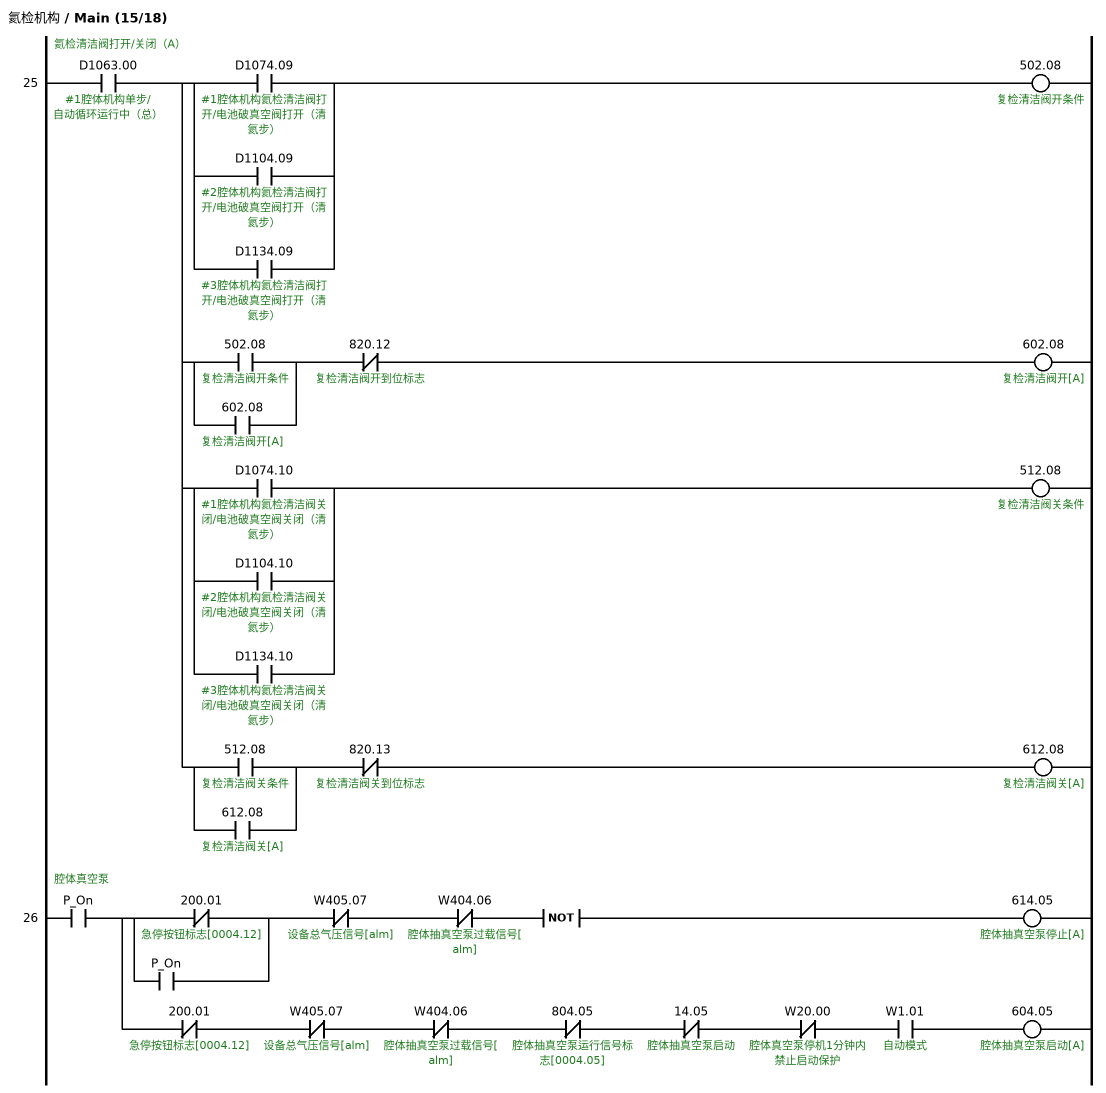
; [picture p144: 氦检机构 / Main, rungs 25-26]
; rung 25: 氦检清洁阀打开/关闭（A）
LD D1063.00  ; #1腔体机构单步/自动循环运行中（总）
OUT TR0
LD D1074.09  ; #1腔体机构氦检清洁阀打开/电池破真空阀打开（清氦步）
OR D1104.09  ; #2腔体机构氦检清洁阀打开/电池破真空阀打开（清氦步）
OR D1134.09  ; #3腔体机构氦检清洁阀打开/电池破真空阀打开（清氦步）
ANDLD
OUT 502.08  ; 复检清洁阀开条件
LD TR0
LD 502.08  ; 复检清洁阀开条件
OR 602.08  ; 复检清洁阀开[A]
ANDLD
ANDNOT 820.12  ; 复检清洁阀开到位标志
OUT 602.08  ; 复检清洁阀开[A]
LD TR0
LD D1074.10  ; #1腔体机构氦检清洁阀关闭/电池破真空阀关闭（清氦步）
OR D1104.10  ; #2腔体机构氦检清洁阀关闭/电池破真空阀关闭（清氦步）
OR D1134.10  ; #3腔体机构氦检清洁阀关闭/电池破真空阀关闭（清氦步）
ANDLD
OUT 512.08  ; 复检清洁阀关条件
LD TR0
LD 512.08  ; 复检清洁阀关条件
OR 612.08  ; 复检清洁阀关[A]
ANDLD
ANDNOT 820.13  ; 复检清洁阀关到位标志
OUT 612.08  ; 复检清洁阀关[A]
; rung 26: 腔体真空泵
LD P_On
OUT TR0
LDNOT 200.01  ; 急停按钮标志[0004.12]
OR P_On
ANDLD
ANDNOT W405.07  ; 设备总气压信号[alm]
ANDNOT W404.06  ; 腔体抽真空泵过载信号[alm]
NOT(520)
OUT 614.05  ; 腔体抽真空泵停止[A]
LD TR0
ANDNOT 200.01  ; 急停按钮标志[0004.12]
ANDNOT W405.07  ; 设备总气压信号[alm]
ANDNOT W404.06  ; 腔体抽真空泵过载信号[alm]
ANDNOT 804.05  ; 腔体抽真空泵运行信号标志[0004.05]
ANDNOT 14.05  ; 腔体抽真空泵启动
ANDNOT W20.00  ; 腔体真空泵停机1分钟内禁止启动保护
AND W1.01  ; 自动模式
OUT 604.05  ; 腔体抽真空泵启动[A]

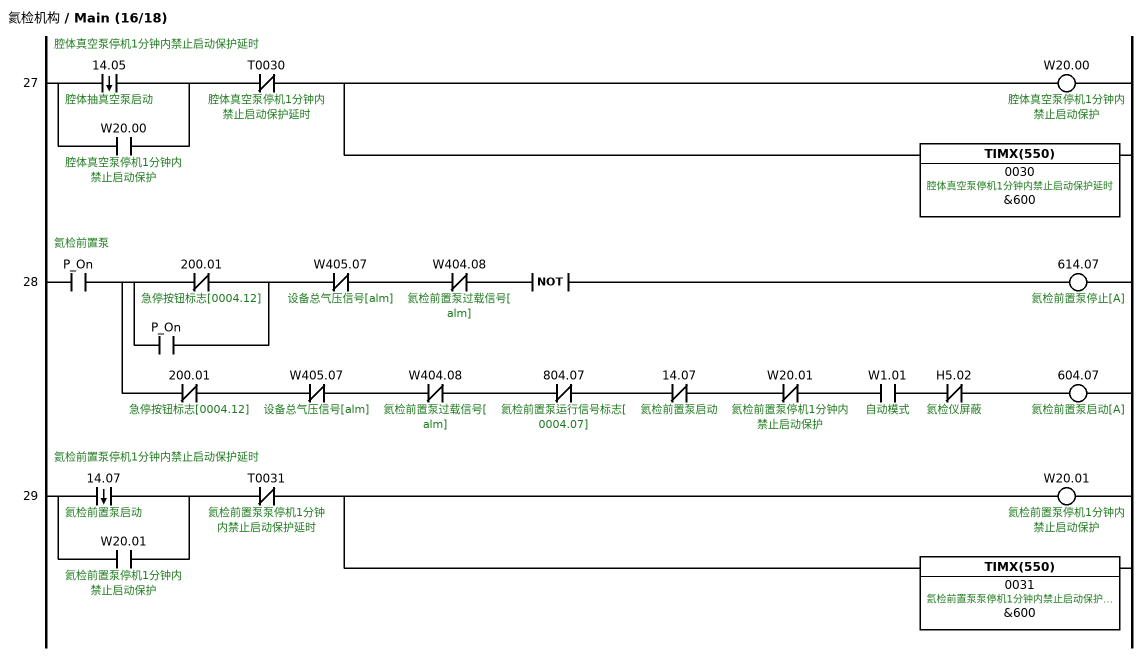
; rung 27: 腔体真空泵停机1分钟内禁止启动保护延时
%LD 14.05  ; 腔体抽真空泵启动
OR W20.00  ; 腔体真空泵停机1分钟内禁止启动保护
ANDNOT T0030  ; 腔体真空泵停机1分钟内禁止启动保护延时
OUT W20.00  ; 腔体真空泵停机1分钟内禁止启动保护
TIMX(550) 0030 &600  ; 腔体真空泵停机1分钟内禁止启动保护延时
; rung 28: 氦检前置泵
LD P_On
OUT TR0
LDNOT 200.01  ; 急停按钮标志[0004.12]
OR P_On
ANDLD
ANDNOT W405.07  ; 设备总气压信号[alm]
ANDNOT W404.08  ; 氦检前置泵过载信号[alm]
NOT(520)
OUT 614.07  ; 氦检前置泵停止[A]
LD TR0
ANDNOT 200.01  ; 急停按钮标志[0004.12]
ANDNOT W405.07  ; 设备总气压信号[alm]
ANDNOT W404.08  ; 氦检前置泵过载信号[alm]
ANDNOT 804.07  ; 氦检前置泵运行信号标志[0004.07]
ANDNOT 14.07  ; 氦检前置泵启动
ANDNOT W20.01  ; 氦检前置泵停机1分钟内禁止启动保护
AND W1.01  ; 自动模式
ANDNOT H5.02  ; 氦检仪屏蔽
OUT 604.07  ; 氦检前置泵启动[A]
; rung 29: 氦检前置泵停机1分钟内禁止启动保护延时
%LD 14.07  ; 氦检前置泵启动
OR W20.01  ; 氦检前置泵停机1分钟内禁止启动保护
ANDNOT T0031  ; 氦检前置泵泵停机1分钟内禁止启动保护延时
OUT W20.01  ; 氦检前置泵停机1分钟内禁止启动保护
TIMX(550) 0031 &600  ; 氦检前置泵泵停机1分钟内禁止启动保护延时

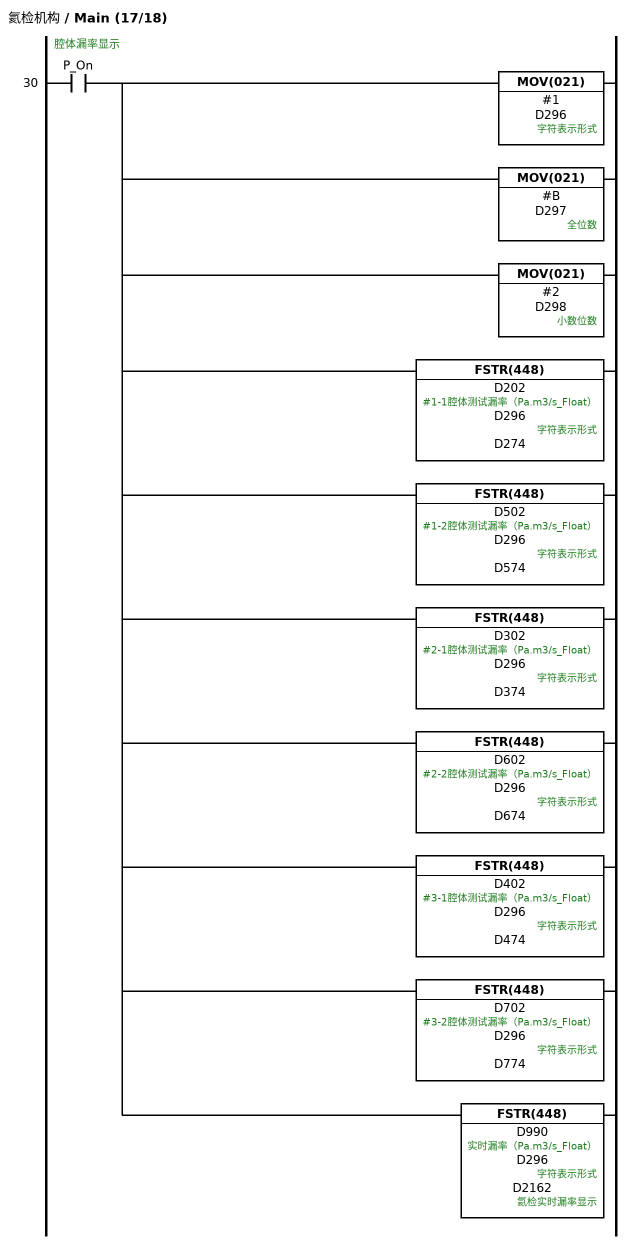
; rung 30: 腔体漏率显示
LD P_On
MOV(021) #1 D296  ; 字符表示形式
MOV(021) #B D297  ; 全位数
MOV(021) #2 D298  ; 小数位数
FSTR(448) D202 D296 D274  ; #1-1腔体测试漏率（Pa.m3/s_Float）, 字符表示形式
FSTR(448) D502 D296 D574  ; #1-2腔体测试漏率（Pa.m3/s_Float）, 字符表示形式
FSTR(448) D302 D296 D374  ; #2-1腔体测试漏率（Pa.m3/s_Float）, 字符表示形式
FSTR(448) D602 D296 D674  ; #2-2腔体测试漏率（Pa.m3/s_Float）, 字符表示形式
FSTR(448) D402 D296 D474  ; #3-1腔体测试漏率（Pa.m3/s_Float）, 字符表示形式
FSTR(448) D702 D296 D774  ; #3-2腔体测试漏率（Pa.m3/s_Float）, 字符表示形式
FSTR(448) D990 D296 D2162  ; 实时漏率（Pa.m3/s_Float）, 字符表示形式, 氦检实时漏率显示

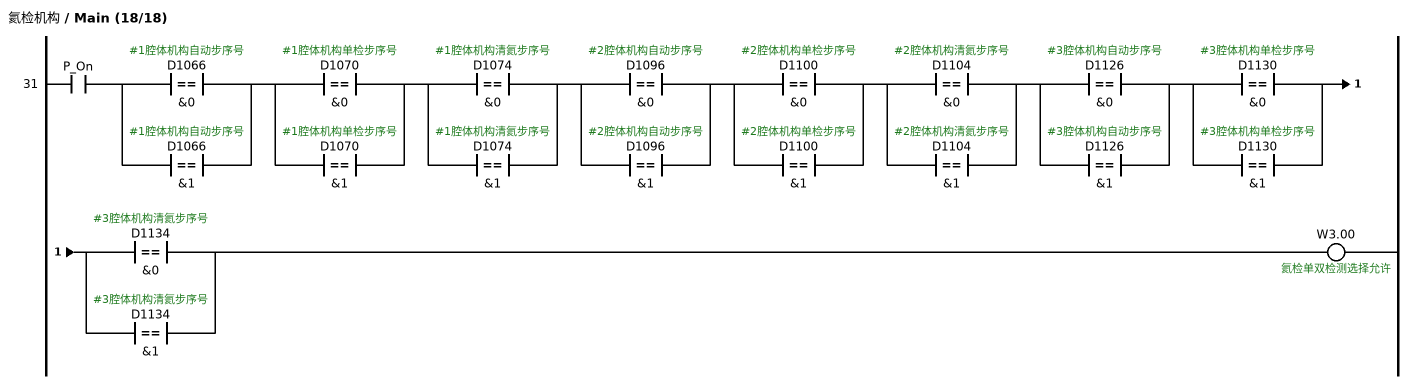
; rung 31
LD P_On
LD=L(301) D1066 &0  ; #1腔体机构自动步序号
OR=L(301) D1066 &1  ; #1腔体机构自动步序号
ANDLD
LD=L(301) D1070 &0  ; #1腔体机构单检步序号
OR=L(301) D1070 &1  ; #1腔体机构单检步序号
ANDLD
LD=L(301) D1074 &0  ; #1腔体机构清氦步序号
OR=L(301) D1074 &1  ; #1腔体机构清氦步序号
ANDLD
LD=L(301) D1096 &0  ; #2腔体机构自动步序号
OR=L(301) D1096 &1  ; #2腔体机构自动步序号
ANDLD
LD=L(301) D1100 &0  ; #2腔体机构单检步序号
OR=L(301) D1100 &1  ; #2腔体机构单检步序号
ANDLD
LD=L(301) D1104 &0  ; #2腔体机构清氦步序号
OR=L(301) D1104 &1  ; #2腔体机构清氦步序号
ANDLD
LD=L(301) D1126 &0  ; #3腔体机构自动步序号
OR=L(301) D1126 &1  ; #3腔体机构自动步序号
ANDLD
LD=L(301) D1130 &0  ; #3腔体机构单检步序号
OR=L(301) D1130 &1  ; #3腔体机构单检步序号
ANDLD
LD=L(301) D1134 &0  ; #3腔体机构清氦步序号
OR=L(301) D1134 &1  ; #3腔体机构清氦步序号
ANDLD
OUT W3.00  ; 氦检单双检测选择允许

### Section 氦检腔1手动

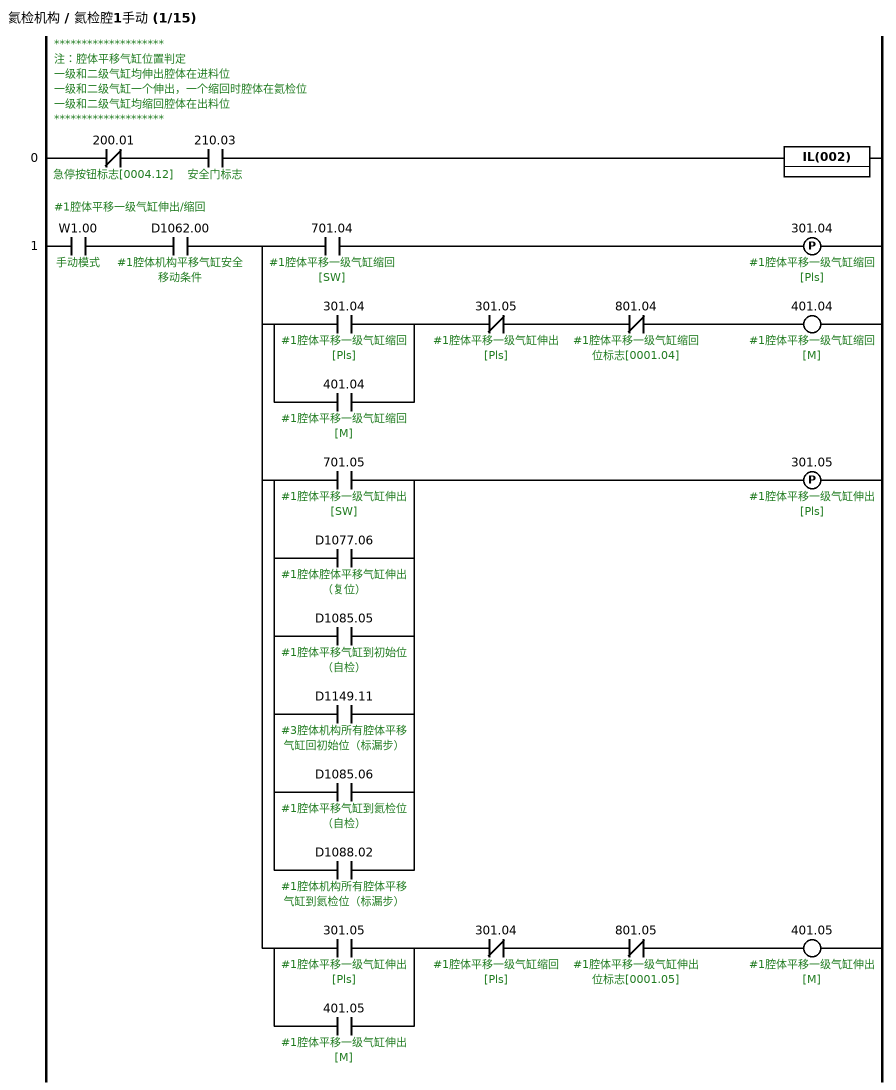
; rung 0: ******************** / 注：腔体平移气缸位置判定 / 一级和二级气缸均伸出腔体在进料位 / 一级和二级气缸一个伸出，一个缩回时腔体在氦检位 / 一级和二级气缸均缩回腔体在出料位 / ********************
LDNOT 200.01  ; 急停按钮标志[0004.12]
AND 210.03  ; 安全门标志
IL(002)
; rung 1: #1腔体平移一级气缸伸出/缩回
LD W1.00  ; 手动模式
AND D1062.00  ; #1腔体机构平移气缸安全移动条件
OUT TR0
AND 701.04  ; #1腔体平移一级气缸缩回[SW]
DIFU(013) 301.04  ; #1腔体平移一级气缸缩回[Pls]
LD TR0
LD 301.04  ; #1腔体平移一级气缸缩回[Pls]
OR 401.04  ; #1腔体平移一级气缸缩回[M]
ANDLD
ANDNOT 301.05  ; #1腔体平移一级气缸伸出[Pls]
ANDNOT 801.04  ; #1腔体平移一级气缸缩回位标志[0001.04]
OUT 401.04  ; #1腔体平移一级气缸缩回[M]
LD TR0
LD 701.05  ; #1腔体平移一级气缸伸出[SW]
OR D1077.06  ; #1腔体腔体平移气缸伸出（复位）
OR D1085.05  ; #1腔体平移气缸到初始位（自检）
OR D1149.11  ; #3腔体机构所有腔体平移气缸回初始位（标漏步）
OR D1085.06  ; #1腔体平移气缸到氦检位（自检）
OR D1088.02  ; #1腔体机构所有腔体平移气缸到氦检位（标漏步）
ANDLD
DIFU(013) 301.05  ; #1腔体平移一级气缸伸出[Pls]
LD TR0
LD 301.05  ; #1腔体平移一级气缸伸出[Pls]
OR 401.05  ; #1腔体平移一级气缸伸出[M]
ANDLD
ANDNOT 301.04  ; #1腔体平移一级气缸缩回[Pls]
ANDNOT 801.05  ; #1腔体平移一级气缸伸出位标志[0001.05]
OUT 401.05  ; #1腔体平移一级气缸伸出[M]

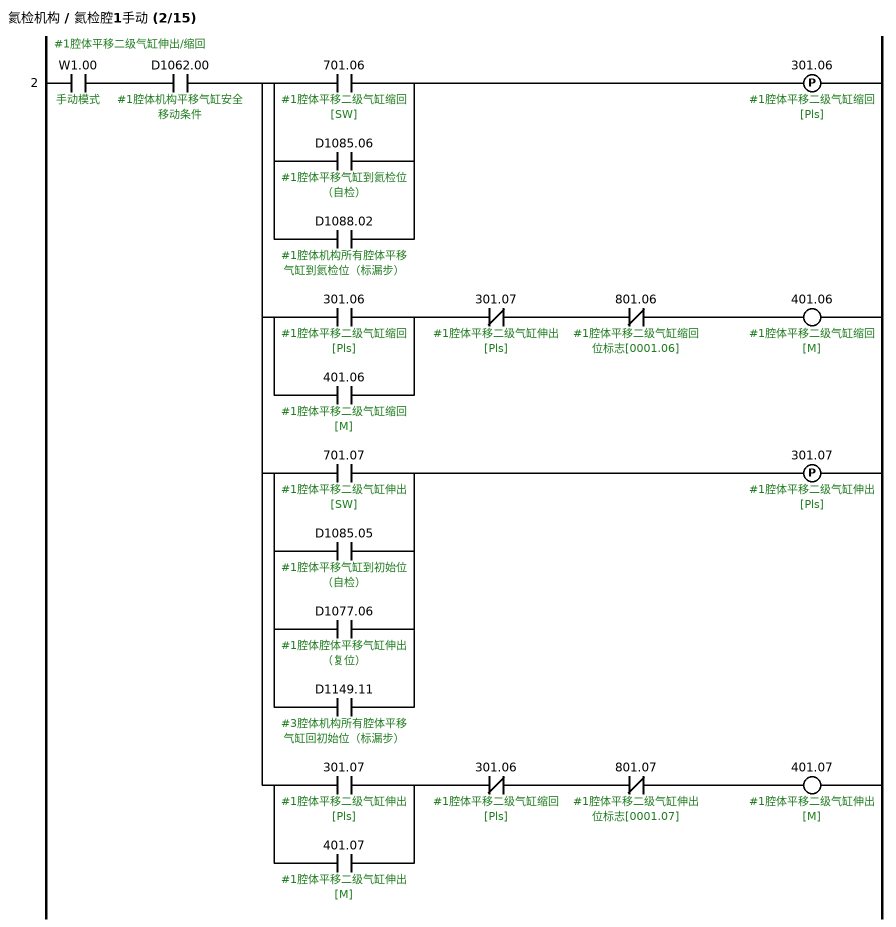
; rung 2: #1腔体平移二级气缸伸出/缩回
LD W1.00  ; 手动模式
AND D1062.00  ; #1腔体机构平移气缸安全移动条件
OUT TR0
LD 701.06  ; #1腔体平移二级气缸缩回[SW]
OR D1085.06  ; #1腔体平移气缸到氦检位（自检）
OR D1088.02  ; #1腔体机构所有腔体平移气缸到氦检位（标漏步）
ANDLD
DIFU(013) 301.06  ; #1腔体平移二级气缸缩回[Pls]
LD TR0
LD 301.06  ; #1腔体平移二级气缸缩回[Pls]
OR 401.06  ; #1腔体平移二级气缸缩回[M]
ANDLD
ANDNOT 301.07  ; #1腔体平移二级气缸伸出[Pls]
ANDNOT 801.06  ; #1腔体平移二级气缸缩回位标志[0001.06]
OUT 401.06  ; #1腔体平移二级气缸缩回[M]
LD TR0
LD 701.07  ; #1腔体平移二级气缸伸出[SW]
OR D1085.05  ; #1腔体平移气缸到初始位（自检）
OR D1077.06  ; #1腔体腔体平移气缸伸出（复位）
OR D1149.11  ; #3腔体机构所有腔体平移气缸回初始位（标漏步）
ANDLD
DIFU(013) 301.07  ; #1腔体平移二级气缸伸出[Pls]
LD TR0
LD 301.07  ; #1腔体平移二级气缸伸出[Pls]
OR 401.07  ; #1腔体平移二级气缸伸出[M]
ANDLD
ANDNOT 301.06  ; #1腔体平移二级气缸缩回[Pls]
ANDNOT 801.07  ; #1腔体平移二级气缸伸出位标志[0001.07]
OUT 401.07  ; #1腔体平移二级气缸伸出[M]

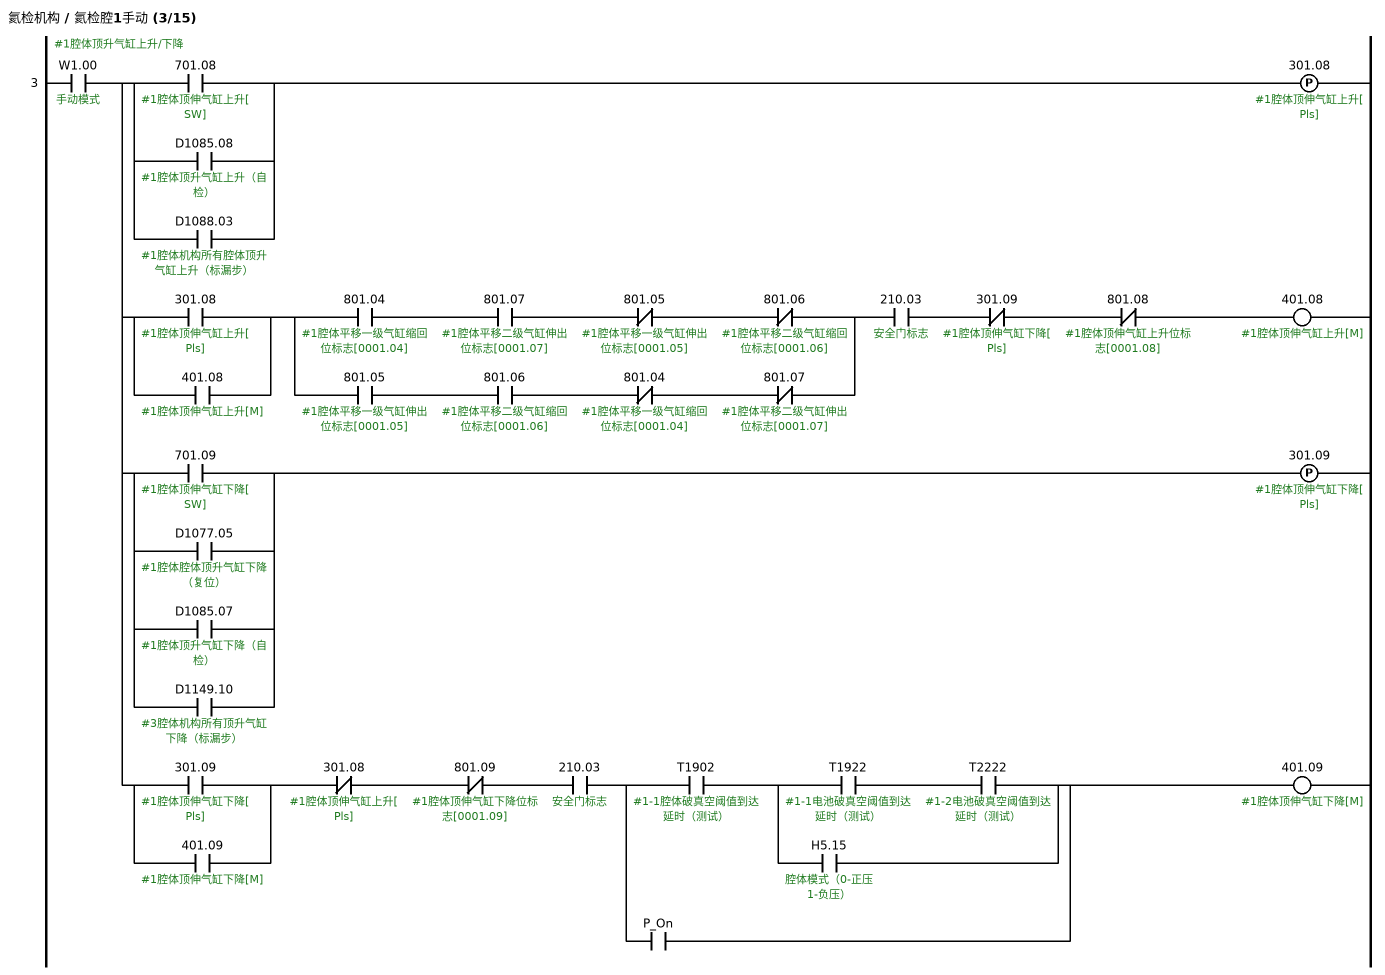
; rung 3: #1腔体顶升气缸上升/下降
LD W1.00  ; 手动模式
OUT TR0
LD 701.08  ; #1腔体顶伸气缸上升[SW]
OR D1085.08  ; #1腔体顶升气缸上升（自检）
OR D1088.03  ; #1腔体机构所有腔体顶升气缸上升（标漏步）
ANDLD
DIFU(013) 301.08  ; #1腔体顶伸气缸上升[Pls]
LD TR0
LD 301.08  ; #1腔体顶伸气缸上升[Pls]
OR 401.08  ; #1腔体顶伸气缸上升[M]
ANDLD
LD 801.04  ; #1腔体平移一级气缸缩回位标志[0001.04]
AND 801.07  ; #1腔体平移二级气缸伸出位标志[0001.07]
ANDNOT 801.05  ; #1腔体平移一级气缸伸出位标志[0001.05]
ANDNOT 801.06  ; #1腔体平移二级气缸缩回位标志[0001.06]
LD 801.05  ; #1腔体平移一级气缸伸出位标志[0001.05]
AND 801.06  ; #1腔体平移二级气缸缩回位标志[0001.06]
ANDNOT 801.04  ; #1腔体平移一级气缸缩回位标志[0001.04]
ANDNOT 801.07  ; #1腔体平移二级气缸伸出位标志[0001.07]
ORLD
ANDLD
AND 210.03  ; 安全门标志
ANDNOT 301.09  ; #1腔体顶伸气缸下降[Pls]
ANDNOT 801.08  ; #1腔体顶伸气缸上升位标志[0001.08]
OUT 401.08  ; #1腔体顶伸气缸上升[M]
LD TR0
LD 701.09  ; #1腔体顶伸气缸下降[SW]
OR D1077.05  ; #1腔体腔体顶升气缸下降（复位）
OR D1085.07  ; #1腔体顶升气缸下降（自检）
OR D1149.10  ; #3腔体机构所有顶升气缸下降（标漏步）
ANDLD
DIFU(013) 301.09  ; #1腔体顶伸气缸下降[Pls]
LD TR0
LD 301.09  ; #1腔体顶伸气缸下降[Pls]
OR 401.09  ; #1腔体顶伸气缸下降[M]
ANDLD
ANDNOT 301.08  ; #1腔体顶伸气缸上升[Pls]
ANDNOT 801.09  ; #1腔体顶伸气缸下降位标志[0001.09]
AND 210.03  ; 安全门标志
LD T1902  ; #1-1腔体破真空阈值到达延时（测试）
LD T1922  ; #1-1电池破真空阈值到达延时（测试）
AND T2222  ; #1-2电池破真空阈值到达延时（测试）
OR H5.15  ; 腔体模式（0-正压 1-负压）
ANDLD
OR P_On
ANDLD
OUT 401.09  ; #1腔体顶伸气缸下降[M]

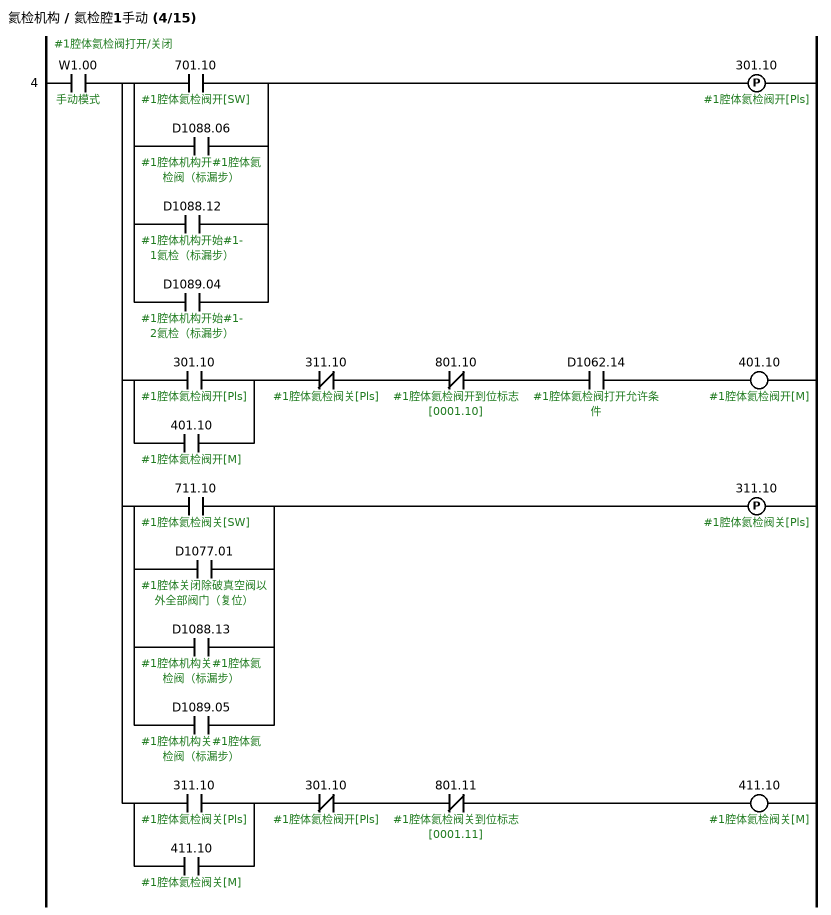
; rung 4: #1腔体氦检阀打开/关闭
LD W1.00  ; 手动模式
OUT TR0
LD 701.10  ; #1腔体氦检阀开[SW]
OR D1088.06  ; #1腔体机构开#1腔体氦检阀（标漏步）
OR D1088.12  ; #1腔体机构开始#1-1氦检（标漏步）
OR D1089.04  ; #1腔体机构开始#1-2氦检（标漏步）
ANDLD
DIFU(013) 301.10  ; #1腔体氦检阀开[Pls]
LD TR0
LD 301.10  ; #1腔体氦检阀开[Pls]
OR 401.10  ; #1腔体氦检阀开[M]
ANDLD
ANDNOT 311.10  ; #1腔体氦检阀关[Pls]
ANDNOT 801.10  ; #1腔体氦检阀开到位标志[0001.10]
AND D1062.14  ; #1腔体氦检阀打开允许条件
OUT 401.10  ; #1腔体氦检阀开[M]
LD TR0
LD 711.10  ; #1腔体氦检阀关[SW]
OR D1077.01  ; #1腔体关闭除破真空阀以外全部阀门（复位）
OR D1088.13  ; #1腔体机构关#1腔体氦检阀（标漏步）
OR D1089.05  ; #1腔体机构关#1腔体氦检阀（标漏步）
ANDLD
DIFU(013) 311.10  ; #1腔体氦检阀关[Pls]
LD TR0
LD 311.10  ; #1腔体氦检阀关[Pls]
OR 411.10  ; #1腔体氦检阀关[M]
ANDLD
ANDNOT 301.10  ; #1腔体氦检阀开[Pls]
ANDNOT 801.11  ; #1腔体氦检阀关到位标志[0001.11]
OUT 411.10  ; #1腔体氦检阀关[M]

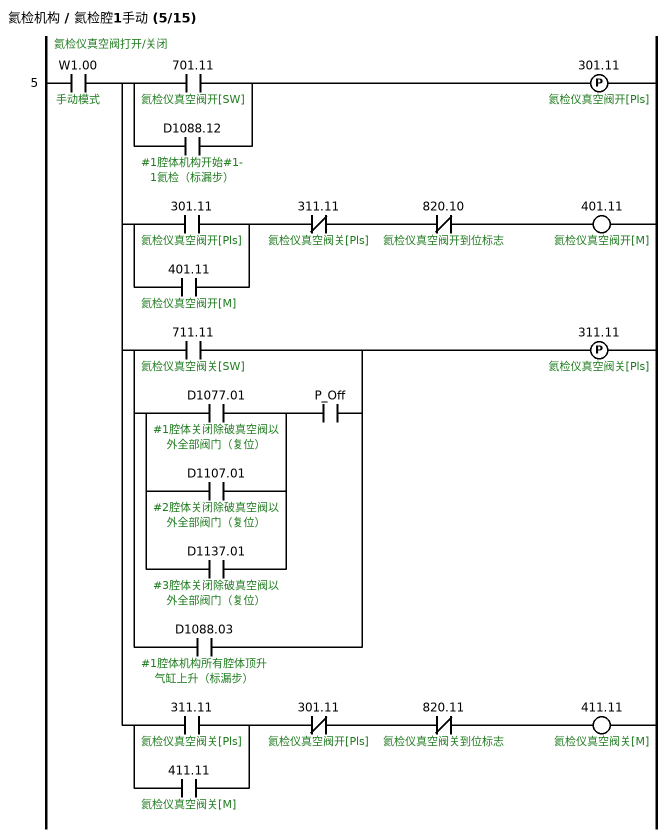
; rung 5: 氦检仪真空阀打开/关闭
LD W1.00  ; 手动模式
OUT TR0
LD 701.11  ; 氦检仪真空阀开[SW]
OR D1088.12  ; #1腔体机构开始#1-1氦检（标漏步）
ANDLD
DIFU(013) 301.11  ; 氦检仪真空阀开[Pls]
LD TR0
LD 301.11  ; 氦检仪真空阀开[Pls]
OR 401.11  ; 氦检仪真空阀开[M]
ANDLD
ANDNOT 311.11  ; 氦检仪真空阀关[Pls]
ANDNOT 820.10  ; 氦检仪真空阀开到位标志
OUT 401.11  ; 氦检仪真空阀开[M]
LD TR0
LD 711.11  ; 氦检仪真空阀关[SW]
LD D1077.01  ; #1腔体关闭除破真空阀以外全部阀门（复位）
OR D1107.01  ; #2腔体关闭除破真空阀以外全部阀门（复位）
OR D1137.01  ; #3腔体关闭除破真空阀以外全部阀门（复位）
AND P_Off
ORLD
OR D1088.03  ; #1腔体机构所有腔体顶升气缸上升（标漏步）
ANDLD
DIFU(013) 311.11  ; 氦检仪真空阀关[Pls]
LD TR0
LD 311.11  ; 氦检仪真空阀关[Pls]
OR 411.11  ; 氦检仪真空阀关[M]
ANDLD
ANDNOT 301.11  ; 氦检仪真空阀开[Pls]
ANDNOT 820.11  ; 氦检仪真空阀关到位标志
OUT 411.11  ; 氦检仪真空阀关[M]

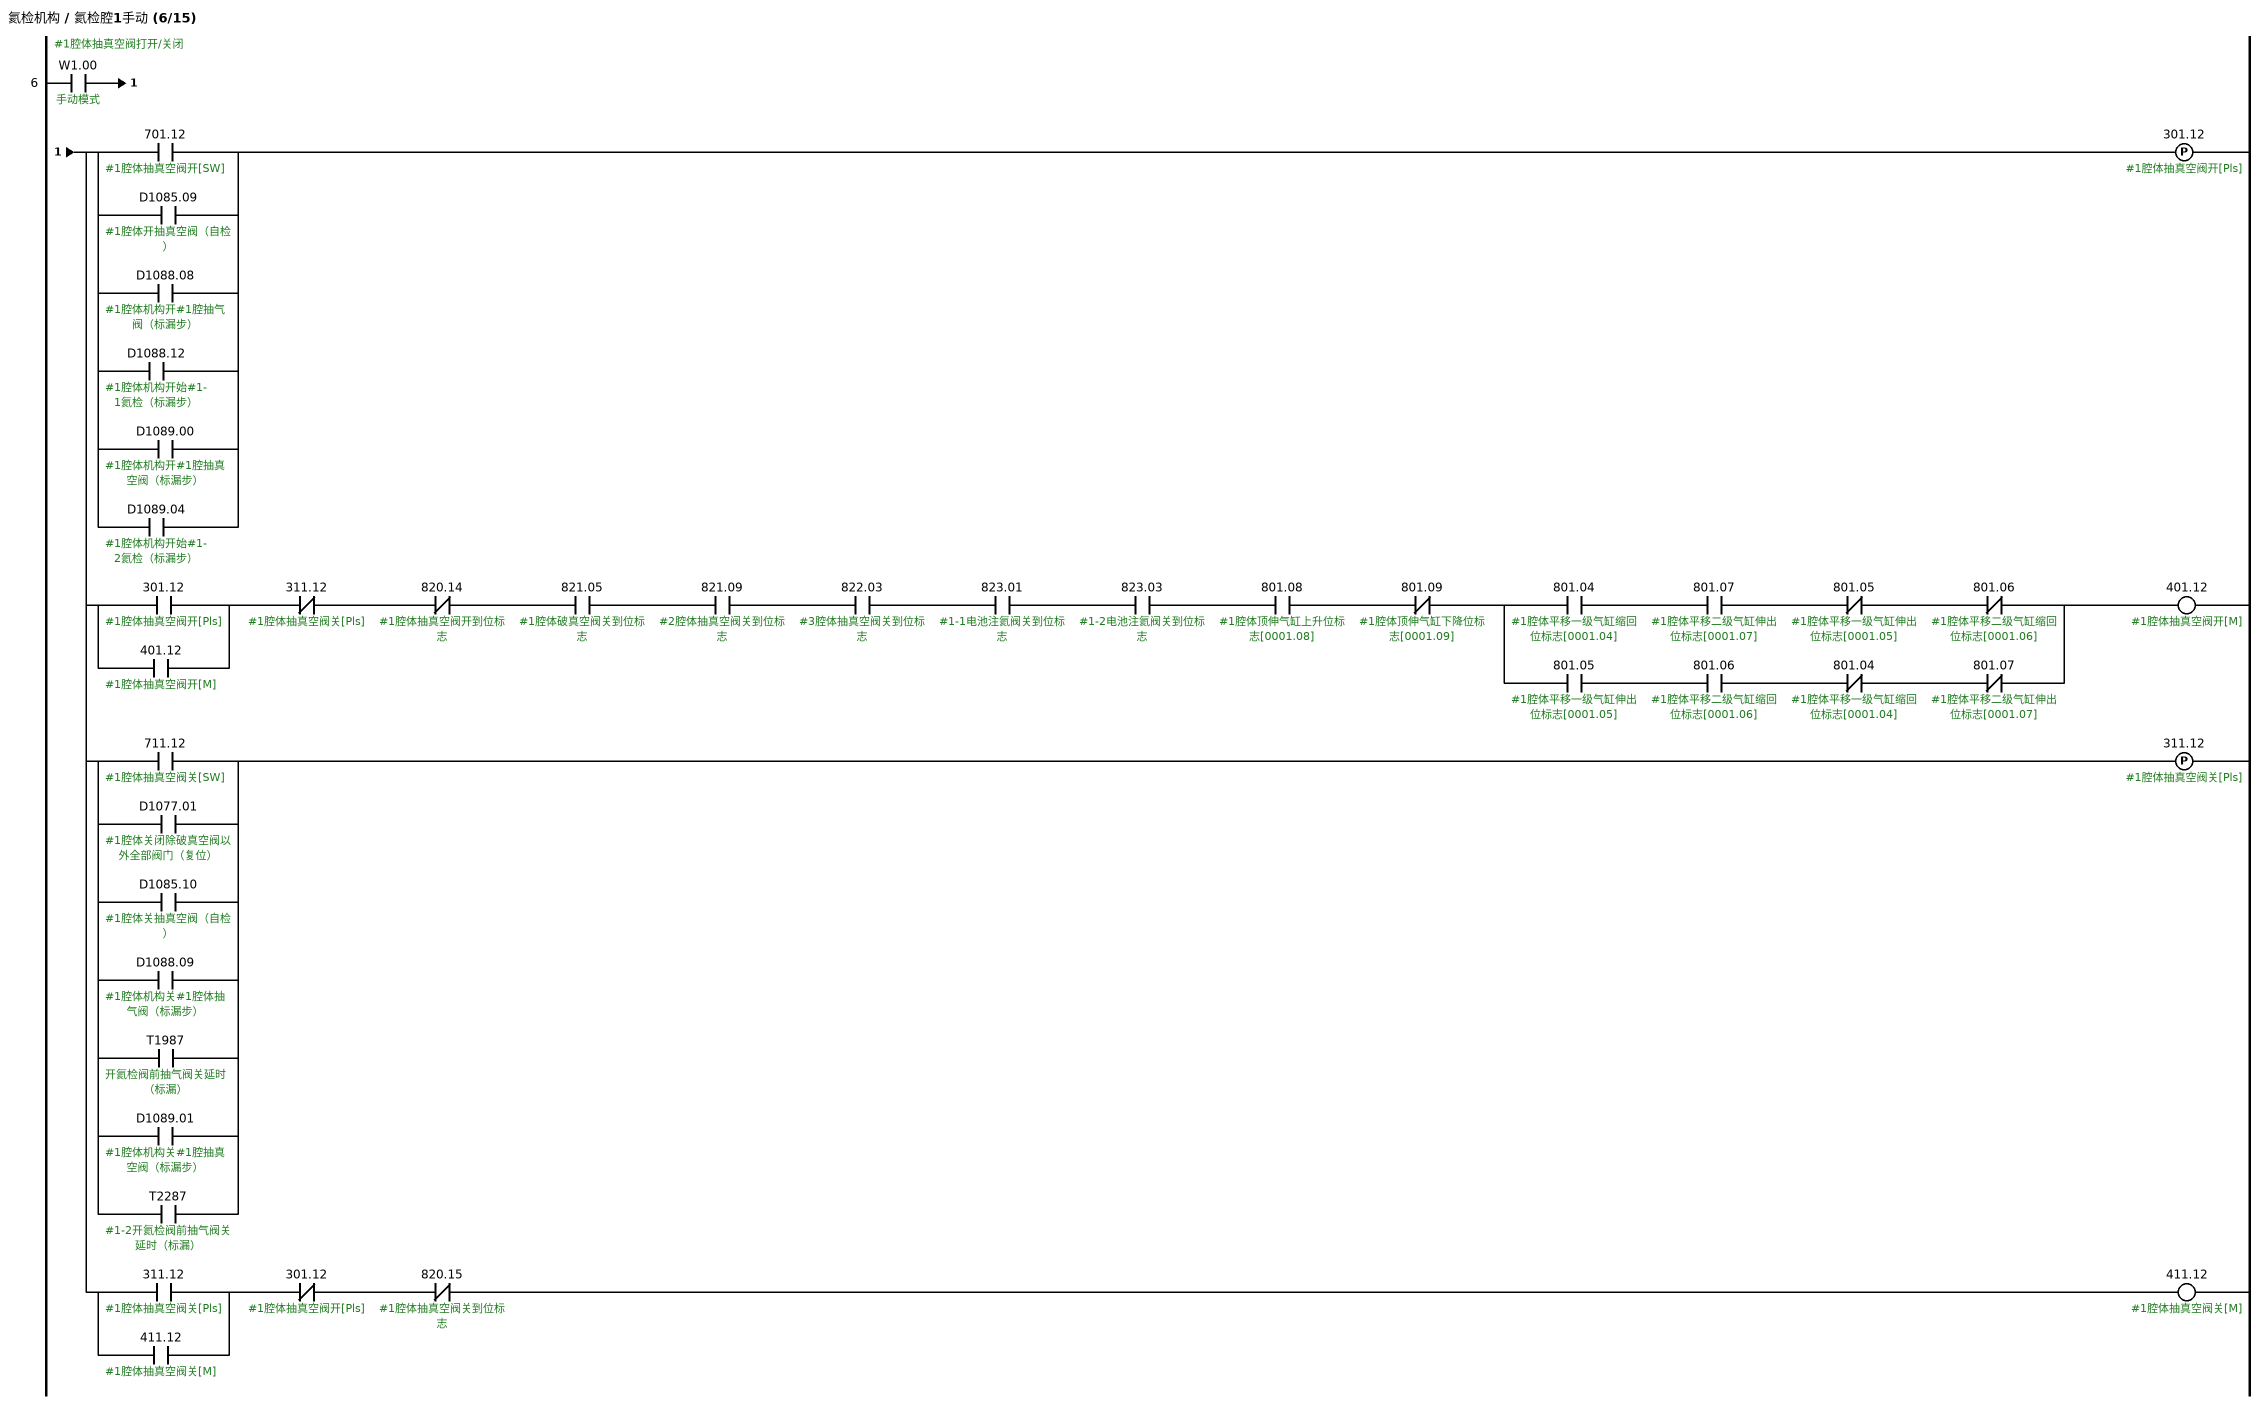
; rung 6: #1腔体抽真空阀打开/关闭
LD W1.00  ; 手动模式
OUT TR0
LD 701.12  ; #1腔体抽真空阀开[SW]
OR D1085.09  ; #1腔体开抽真空阀（自检）
OR D1088.08  ; #1腔体机构开#1腔抽气阀（标漏步）
OR D1088.12  ; #1腔体机构开始#1-1氦检（标漏步）
OR D1089.00  ; #1腔体机构开#1腔抽真空阀（标漏步）
OR D1089.04  ; #1腔体机构开始#1-2氦检（标漏步）
ANDLD
DIFU(013) 301.12  ; #1腔体抽真空阀开[Pls]
LD TR0
LD 301.12  ; #1腔体抽真空阀开[Pls]
OR 401.12  ; #1腔体抽真空阀开[M]
ANDLD
ANDNOT 311.12  ; #1腔体抽真空阀关[Pls]
ANDNOT 820.14  ; #1腔体抽真空阀开到位标志
AND 821.05  ; #1腔体破真空阀关到位标志
AND 821.09  ; #2腔体抽真空阀关到位标志
AND 822.03  ; #3腔体抽真空阀关到位标志
AND 823.01  ; #1-1电池注氦阀关到位标志
AND 823.03  ; #1-2电池注氦阀关到位标志
AND 801.08  ; #1腔体顶伸气缸上升位标志[0001.08]
ANDNOT 801.09  ; #1腔体顶伸气缸下降位标志[0001.09]
LD 801.04  ; #1腔体平移一级气缸缩回位标志[0001.04]
AND 801.07  ; #1腔体平移二级气缸伸出位标志[0001.07]
ANDNOT 801.05  ; #1腔体平移一级气缸伸出位标志[0001.05]
ANDNOT 801.06  ; #1腔体平移二级气缸缩回位标志[0001.06]
LD 801.05  ; #1腔体平移一级气缸伸出位标志[0001.05]
AND 801.06  ; #1腔体平移二级气缸缩回位标志[0001.06]
ANDNOT 801.04  ; #1腔体平移一级气缸缩回位标志[0001.04]
ANDNOT 801.07  ; #1腔体平移二级气缸伸出位标志[0001.07]
ORLD
ANDLD
OUT 401.12  ; #1腔体抽真空阀开[M]
LD TR0
LD 711.12  ; #1腔体抽真空阀关[SW]
OR D1077.01  ; #1腔体关闭除破真空阀以外全部阀门（复位）
OR D1085.10  ; #1腔体关抽真空阀（自检）
OR D1088.09  ; #1腔体机构关#1腔体抽气阀（标漏步）
OR T1987  ; 开氦检阀前抽气阀关延时（标漏）
OR D1089.01  ; #1腔体机构关#1腔抽真空阀（标漏步）
OR T2287  ; #1-2开氦检阀前抽气阀关延时（标漏）
ANDLD
DIFU(013) 311.12  ; #1腔体抽真空阀关[Pls]
LD TR0
LD 311.12  ; #1腔体抽真空阀关[Pls]
OR 411.12  ; #1腔体抽真空阀关[M]
ANDLD
ANDNOT 301.12  ; #1腔体抽真空阀开[Pls]
ANDNOT 820.15  ; #1腔体抽真空阀关到位标志
OUT 411.12  ; #1腔体抽真空阀关[M]

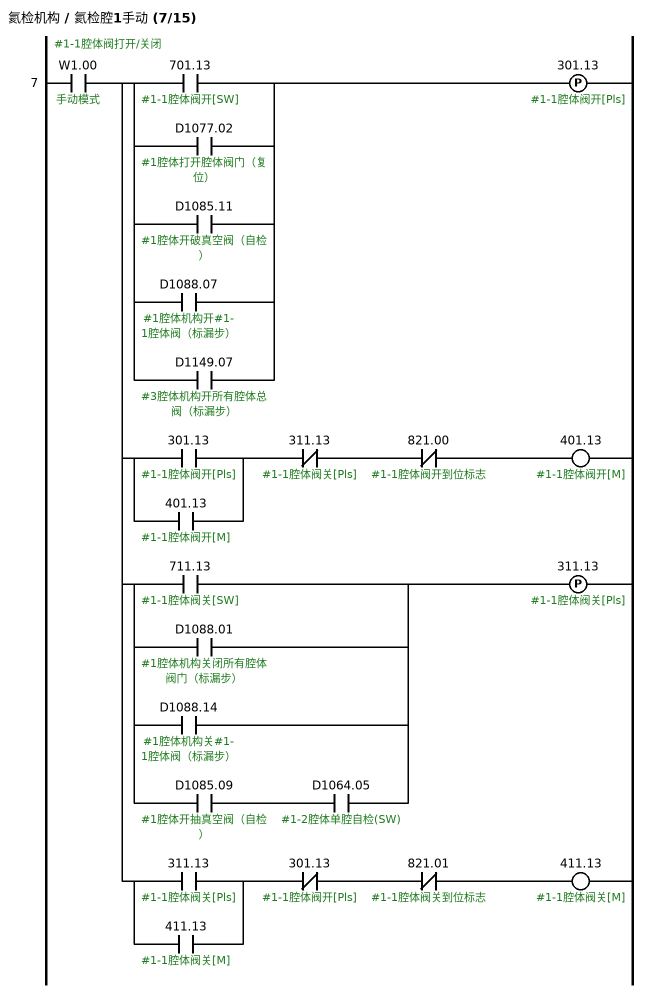
; rung 7: #1-1腔体阀打开/关闭
LD W1.00  ; 手动模式
OUT TR0
LD 701.13  ; #1-1腔体阀开[SW]
OR D1077.02  ; #1腔体打开腔体阀门（复位）
OR D1085.11  ; #1腔体开破真空阀（自检）
OR D1088.07  ; #1腔体机构开#1-1腔体阀（标漏步）
OR D1149.07  ; #3腔体机构开所有腔体总阀（标漏步）
ANDLD
DIFU(013) 301.13  ; #1-1腔体阀开[Pls]
LD TR0
LD 301.13  ; #1-1腔体阀开[Pls]
OR 401.13  ; #1-1腔体阀开[M]
ANDLD
ANDNOT 311.13  ; #1-1腔体阀关[Pls]
ANDNOT 821.00  ; #1-1腔体阀开到位标志
OUT 401.13  ; #1-1腔体阀开[M]
LD TR0
LD 711.13  ; #1-1腔体阀关[SW]
OR D1088.01  ; #1腔体机构关闭所有腔体阀门（标漏步）
OR D1088.14  ; #1腔体机构关#1-1腔体阀（标漏步）
LD D1085.09  ; #1腔体开抽真空阀（自检）
AND D1064.05  ; #1-2腔体单腔自检(SW)
ORLD
ANDLD
DIFU(013) 311.13  ; #1-1腔体阀关[Pls]
LD TR0
LD 311.13  ; #1-1腔体阀关[Pls]
OR 411.13  ; #1-1腔体阀关[M]
ANDLD
ANDNOT 301.13  ; #1-1腔体阀开[Pls]
ANDNOT 821.01  ; #1-1腔体阀关到位标志
OUT 411.13  ; #1-1腔体阀关[M]

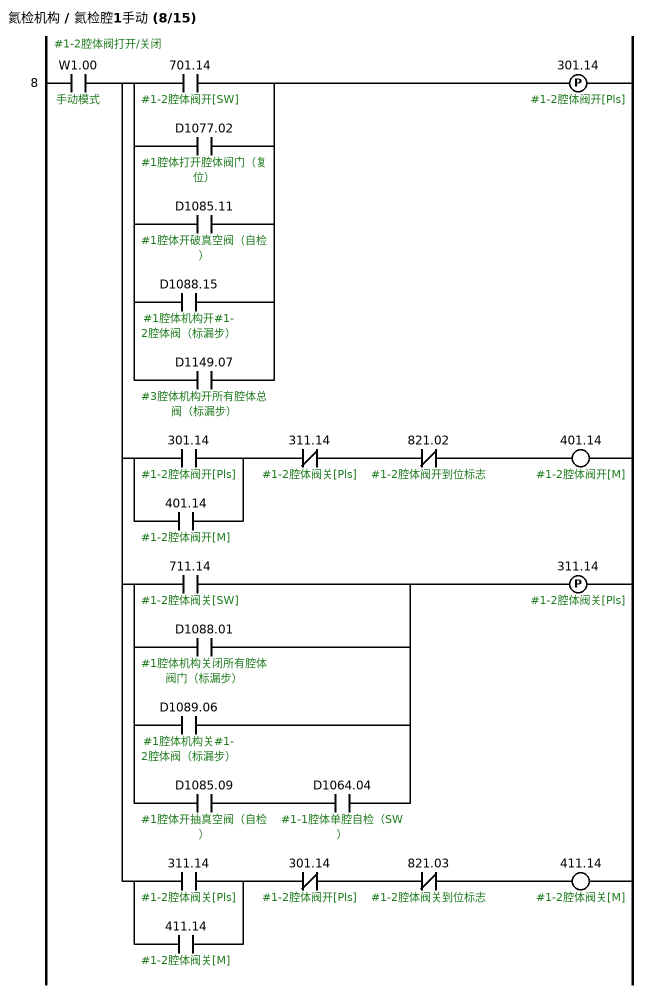
; rung 8: #1-2腔体阀打开/关闭
LD W1.00  ; 手动模式
OUT TR0
LD 701.14  ; #1-2腔体阀开[SW]
OR D1077.02  ; #1腔体打开腔体阀门（复位）
OR D1085.11  ; #1腔体开破真空阀（自检）
OR D1088.15  ; #1腔体机构开#1-2腔体阀（标漏步）
OR D1149.07  ; #3腔体机构开所有腔体总阀（标漏步）
ANDLD
DIFU(013) 301.14  ; #1-2腔体阀开[Pls]
LD TR0
LD 301.14  ; #1-2腔体阀开[Pls]
OR 401.14  ; #1-2腔体阀开[M]
ANDLD
ANDNOT 311.14  ; #1-2腔体阀关[Pls]
ANDNOT 821.02  ; #1-2腔体阀开到位标志
OUT 401.14  ; #1-2腔体阀开[M]
LD TR0
LD 711.14  ; #1-2腔体阀关[SW]
OR D1088.01  ; #1腔体机构关闭所有腔体阀门（标漏步）
OR D1089.06  ; #1腔体机构关#1-2腔体阀（标漏步）
LD D1085.09  ; #1腔体开抽真空阀（自检）
AND D1064.04  ; #1-1腔体单腔自检（SW）
ORLD
ANDLD
DIFU(013) 311.14  ; #1-2腔体阀关[Pls]
LD TR0
LD 311.14  ; #1-2腔体阀关[Pls]
OR 411.14  ; #1-2腔体阀关[M]
ANDLD
ANDNOT 301.14  ; #1-2腔体阀开[Pls]
ANDNOT 821.03  ; #1-2腔体阀关到位标志
OUT 411.14  ; #1-2腔体阀关[M]

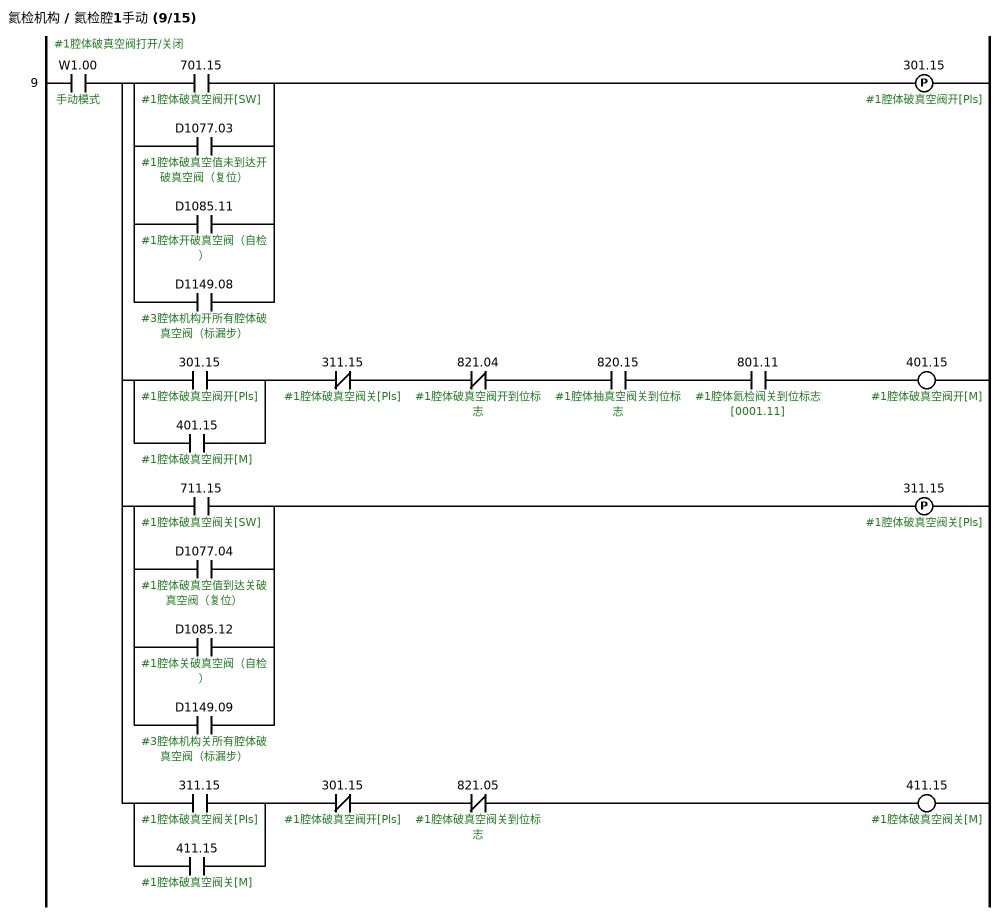
; rung 9: #1腔体破真空阀打开/关闭
LD W1.00  ; 手动模式
OUT TR0
LD 701.15  ; #1腔体破真空阀开[SW]
OR D1077.03  ; #1腔体破真空值未到达开破真空阀（复位）
OR D1085.11  ; #1腔体开破真空阀（自检）
OR D1149.08  ; #3腔体机构开所有腔体破真空阀（标漏步）
ANDLD
DIFU(013) 301.15  ; #1腔体破真空阀开[Pls]
LD TR0
LD 301.15  ; #1腔体破真空阀开[Pls]
OR 401.15  ; #1腔体破真空阀开[M]
ANDLD
ANDNOT 311.15  ; #1腔体破真空阀关[Pls]
ANDNOT 821.04  ; #1腔体破真空阀开到位标志
AND 820.15  ; #1腔体抽真空阀关到位标志
AND 801.11  ; #1腔体氦检阀关到位标志[0001.11]
OUT 401.15  ; #1腔体破真空阀开[M]
LD TR0
LD 711.15  ; #1腔体破真空阀关[SW]
OR D1077.04  ; #1腔体破真空值到达关破真空阀（复位）
OR D1085.12  ; #1腔体关破真空阀（自检）
OR D1149.09  ; #3腔体机构关所有腔体破真空阀（标漏步）
ANDLD
DIFU(013) 311.15  ; #1腔体破真空阀关[Pls]
LD TR0
LD 311.15  ; #1腔体破真空阀关[Pls]
OR 411.15  ; #1腔体破真空阀关[M]
ANDLD
ANDNOT 301.15  ; #1腔体破真空阀开[Pls]
ANDNOT 821.05  ; #1腔体破真空阀关到位标志
OUT 411.15  ; #1腔体破真空阀关[M]

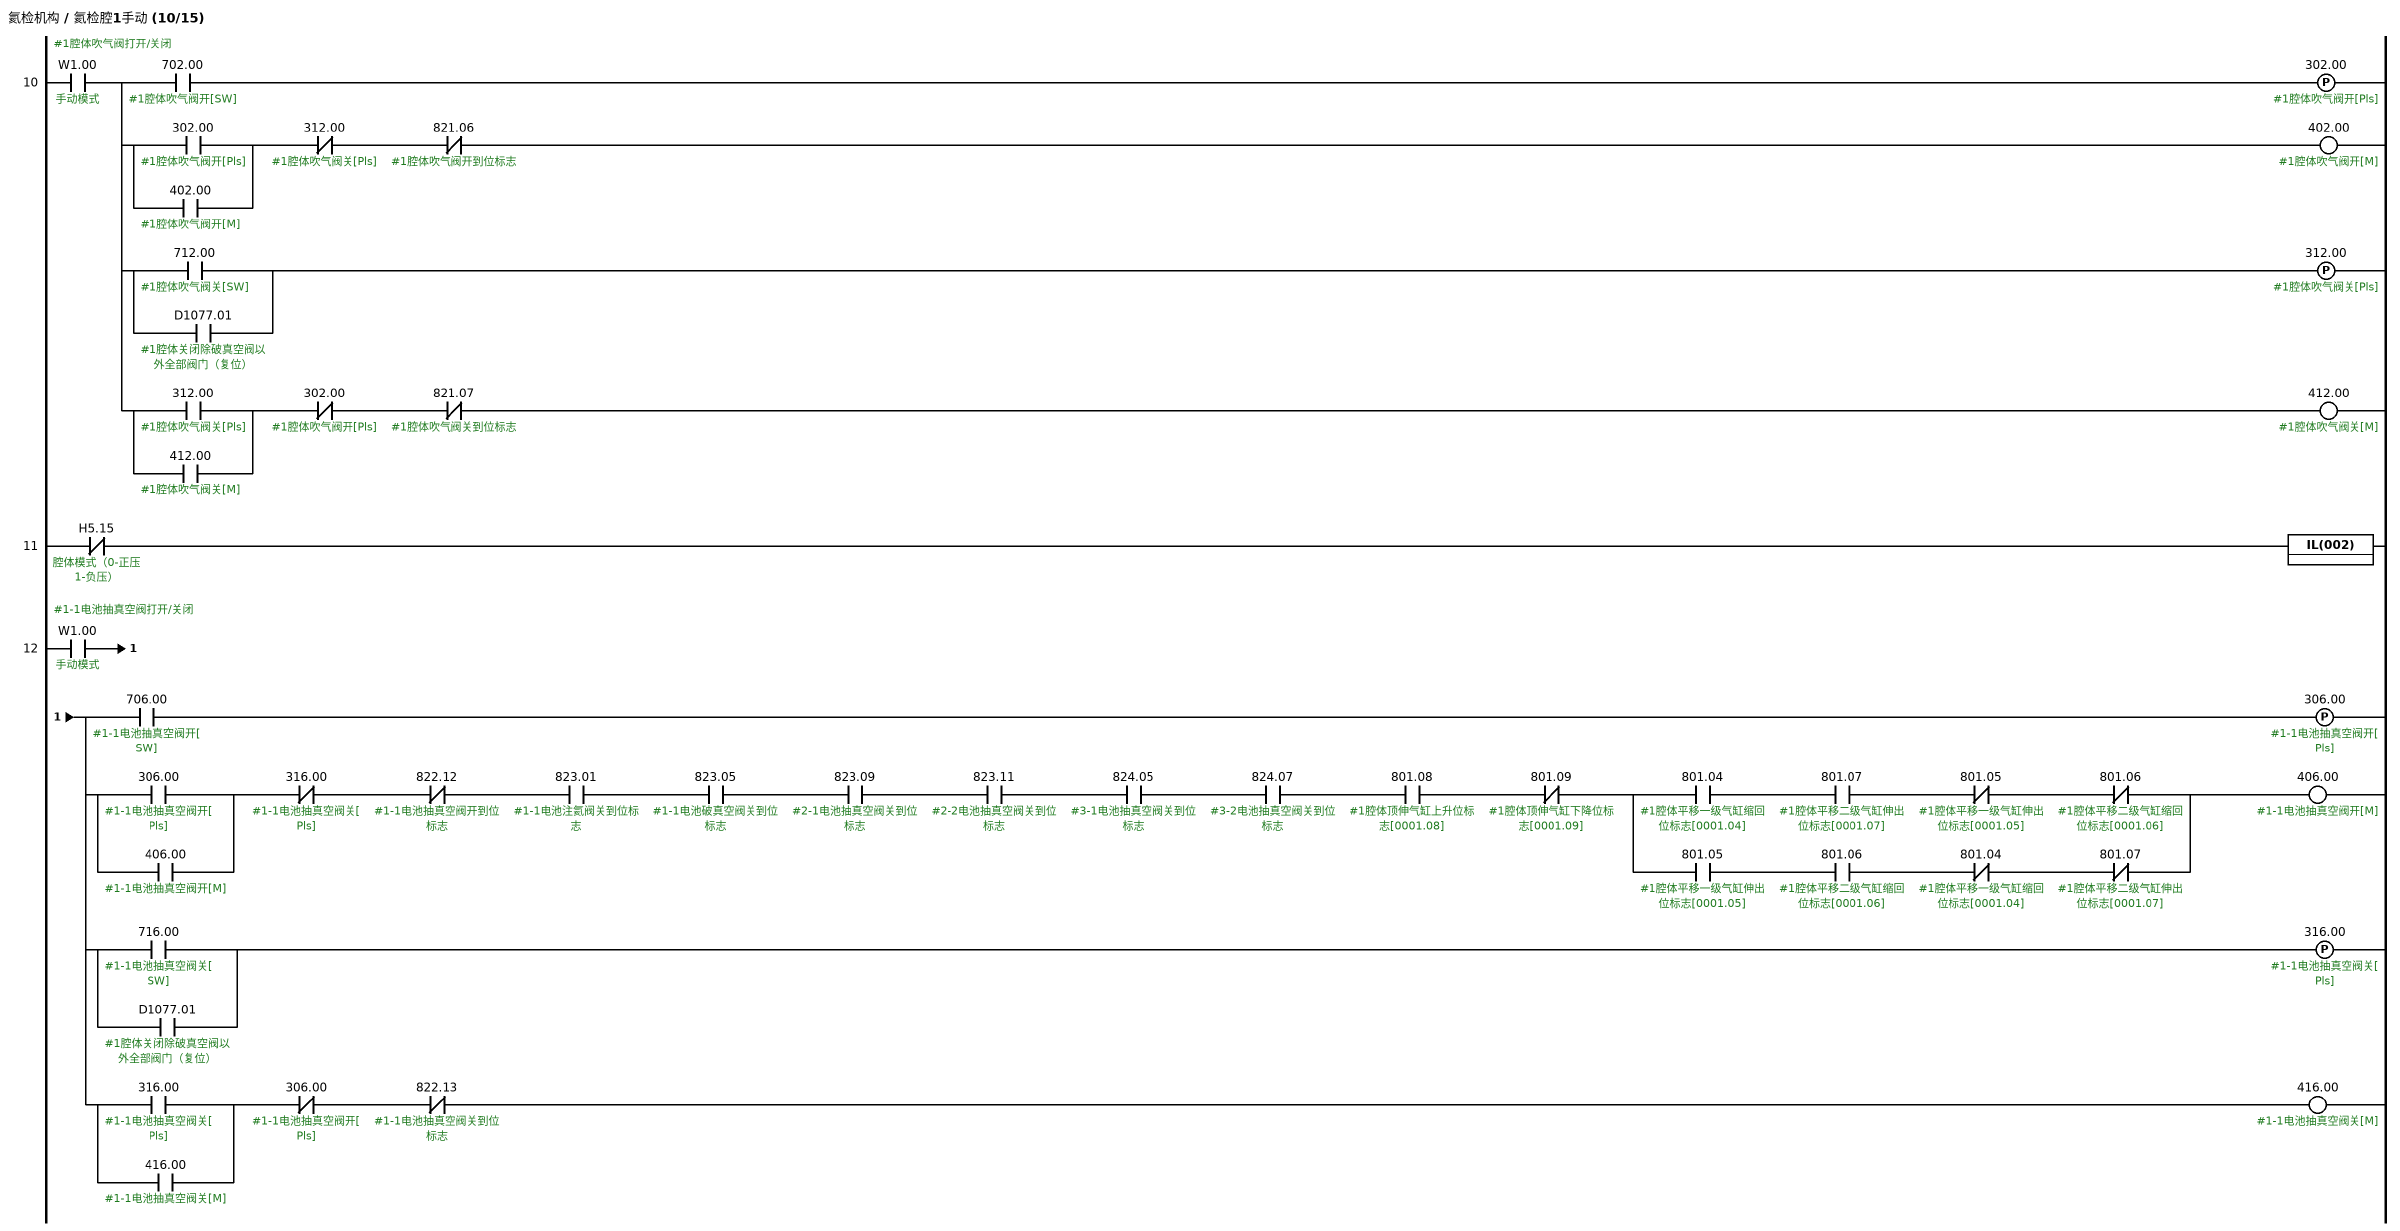
; rung 10: #1腔体吹气阀打开/关闭
LD W1.00  ; 手动模式
OUT TR0
AND 702.00  ; #1腔体吹气阀开[SW]
DIFU(013) 302.00  ; #1腔体吹气阀开[Pls]
LD TR0
LD 302.00  ; #1腔体吹气阀开[Pls]
OR 402.00  ; #1腔体吹气阀开[M]
ANDLD
ANDNOT 312.00  ; #1腔体吹气阀关[Pls]
ANDNOT 821.06  ; #1腔体吹气阀开到位标志
OUT 402.00  ; #1腔体吹气阀开[M]
LD TR0
LD 712.00  ; #1腔体吹气阀关[SW]
OR D1077.01  ; #1腔体关闭除破真空阀以外全部阀门（复位）
ANDLD
DIFU(013) 312.00  ; #1腔体吹气阀关[Pls]
LD TR0
LD 312.00  ; #1腔体吹气阀关[Pls]
OR 412.00  ; #1腔体吹气阀关[M]
ANDLD
ANDNOT 302.00  ; #1腔体吹气阀开[Pls]
ANDNOT 821.07  ; #1腔体吹气阀关到位标志
OUT 412.00  ; #1腔体吹气阀关[M]
; rung 11
LDNOT H5.15  ; 腔体模式（0-正压 1-负压）
IL(002)
; rung 12: #1-1电池抽真空阀打开/关闭
LD W1.00  ; 手动模式
OUT TR0
AND 706.00  ; #1-1电池抽真空阀开[SW]
DIFU(013) 306.00  ; #1-1电池抽真空阀开[Pls]
LD TR0
LD 306.00  ; #1-1电池抽真空阀开[Pls]
OR 406.00  ; #1-1电池抽真空阀开[M]
ANDLD
ANDNOT 316.00  ; #1-1电池抽真空阀关[Pls]
ANDNOT 822.12  ; #1-1电池抽真空阀开到位标志
AND 823.01  ; #1-1电池注氦阀关到位标志
AND 823.05  ; #1-1电池破真空阀关到位标志
AND 823.09  ; #2-1电池抽真空阀关到位标志
AND 823.11  ; #2-2电池抽真空阀关到位标志
AND 824.05  ; #3-1电池抽真空阀关到位标志
AND 824.07  ; #3-2电池抽真空阀关到位标志
AND 801.08  ; #1腔体顶伸气缸上升位标志[0001.08]
ANDNOT 801.09  ; #1腔体顶伸气缸下降位标志[0001.09]
LD 801.04  ; #1腔体平移一级气缸缩回位标志[0001.04]
AND 801.07  ; #1腔体平移二级气缸伸出位标志[0001.07]
ANDNOT 801.05  ; #1腔体平移一级气缸伸出位标志[0001.05]
ANDNOT 801.06  ; #1腔体平移二级气缸缩回位标志[0001.06]
LD 801.05  ; #1腔体平移一级气缸伸出位标志[0001.05]
AND 801.06  ; #1腔体平移二级气缸缩回位标志[0001.06]
ANDNOT 801.04  ; #1腔体平移一级气缸缩回位标志[0001.04]
ANDNOT 801.07  ; #1腔体平移二级气缸伸出位标志[0001.07]
ORLD
ANDLD
OUT 406.00  ; #1-1电池抽真空阀开[M]
LD TR0
LD 716.00  ; #1-1电池抽真空阀关[SW]
OR D1077.01  ; #1腔体关闭除破真空阀以外全部阀门（复位）
ANDLD
DIFU(013) 316.00  ; #1-1电池抽真空阀关[Pls]
LD TR0
LD 316.00  ; #1-1电池抽真空阀关[Pls]
OR 416.00  ; #1-1电池抽真空阀关[M]
ANDLD
ANDNOT 306.00  ; #1-1电池抽真空阀开[Pls]
ANDNOT 822.13  ; #1-1电池抽真空阀关到位标志
OUT 416.00  ; #1-1电池抽真空阀关[M]

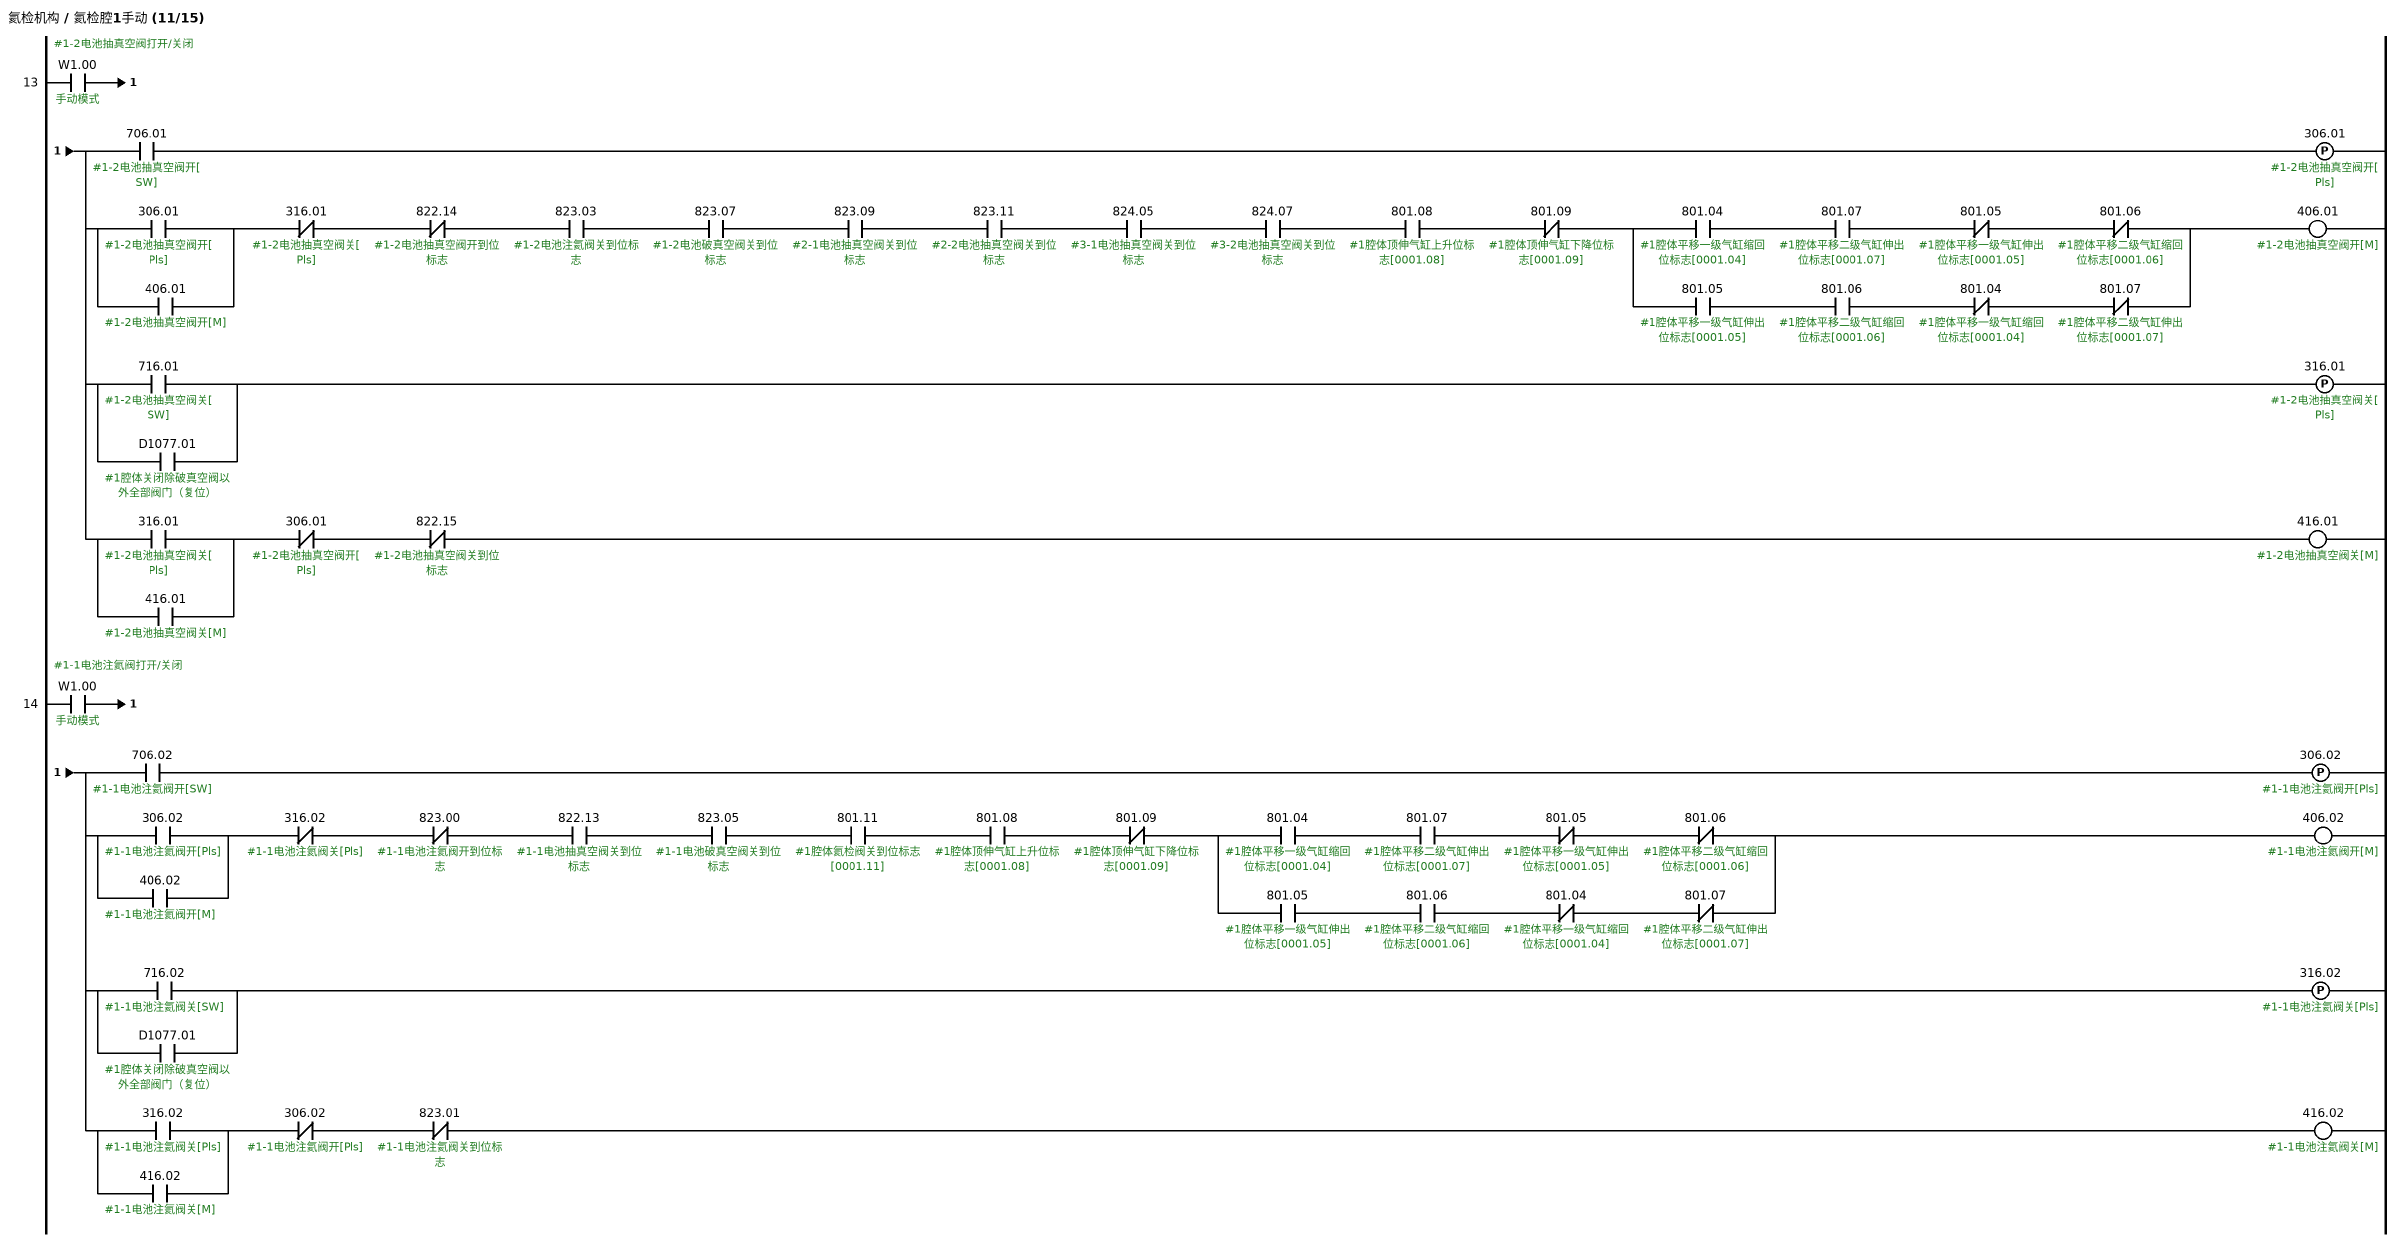
; rung 13: #1-2电池抽真空阀打开/关闭
LD W1.00  ; 手动模式
OUT TR0
AND 706.01  ; #1-2电池抽真空阀开[SW]
DIFU(013) 306.01  ; #1-2电池抽真空阀开[Pls]
LD TR0
LD 306.01  ; #1-2电池抽真空阀开[Pls]
OR 406.01  ; #1-2电池抽真空阀开[M]
ANDLD
ANDNOT 316.01  ; #1-2电池抽真空阀关[Pls]
ANDNOT 822.14  ; #1-2电池抽真空阀开到位标志
AND 823.03  ; #1-2电池注氦阀关到位标志
AND 823.07  ; #1-2电池破真空阀关到位标志
AND 823.09  ; #2-1电池抽真空阀关到位标志
AND 823.11  ; #2-2电池抽真空阀关到位标志
AND 824.05  ; #3-1电池抽真空阀关到位标志
AND 824.07  ; #3-2电池抽真空阀关到位标志
AND 801.08  ; #1腔体顶伸气缸上升位标志[0001.08]
ANDNOT 801.09  ; #1腔体顶伸气缸下降位标志[0001.09]
LD 801.04  ; #1腔体平移一级气缸缩回位标志[0001.04]
AND 801.07  ; #1腔体平移二级气缸伸出位标志[0001.07]
ANDNOT 801.05  ; #1腔体平移一级气缸伸出位标志[0001.05]
ANDNOT 801.06  ; #1腔体平移二级气缸缩回位标志[0001.06]
LD 801.05  ; #1腔体平移一级气缸伸出位标志[0001.05]
AND 801.06  ; #1腔体平移二级气缸缩回位标志[0001.06]
ANDNOT 801.04  ; #1腔体平移一级气缸缩回位标志[0001.04]
ANDNOT 801.07  ; #1腔体平移二级气缸伸出位标志[0001.07]
ORLD
ANDLD
OUT 406.01  ; #1-2电池抽真空阀开[M]
LD TR0
LD 716.01  ; #1-2电池抽真空阀关[SW]
OR D1077.01  ; #1腔体关闭除破真空阀以外全部阀门（复位）
ANDLD
DIFU(013) 316.01  ; #1-2电池抽真空阀关[Pls]
LD TR0
LD 316.01  ; #1-2电池抽真空阀关[Pls]
OR 416.01  ; #1-2电池抽真空阀关[M]
ANDLD
ANDNOT 306.01  ; #1-2电池抽真空阀开[Pls]
ANDNOT 822.15  ; #1-2电池抽真空阀关到位标志
OUT 416.01  ; #1-2电池抽真空阀关[M]
; rung 14: #1-1电池注氦阀打开/关闭
LD W1.00  ; 手动模式
OUT TR0
AND 706.02  ; #1-1电池注氦阀开[SW]
DIFU(013) 306.02  ; #1-1电池注氦阀开[Pls]
LD TR0
LD 306.02  ; #1-1电池注氦阀开[Pls]
OR 406.02  ; #1-1电池注氦阀开[M]
ANDLD
ANDNOT 316.02  ; #1-1电池注氦阀关[Pls]
ANDNOT 823.00  ; #1-1电池注氦阀开到位标志
AND 822.13  ; #1-1电池抽真空阀关到位标志
AND 823.05  ; #1-1电池破真空阀关到位标志
AND 801.11  ; #1腔体氦检阀关到位标志[0001.11]
AND 801.08  ; #1腔体顶伸气缸上升位标志[0001.08]
ANDNOT 801.09  ; #1腔体顶伸气缸下降位标志[0001.09]
LD 801.04  ; #1腔体平移一级气缸缩回位标志[0001.04]
AND 801.07  ; #1腔体平移二级气缸伸出位标志[0001.07]
ANDNOT 801.05  ; #1腔体平移一级气缸伸出位标志[0001.05]
ANDNOT 801.06  ; #1腔体平移二级气缸缩回位标志[0001.06]
LD 801.05  ; #1腔体平移一级气缸伸出位标志[0001.05]
AND 801.06  ; #1腔体平移二级气缸缩回位标志[0001.06]
ANDNOT 801.04  ; #1腔体平移一级气缸缩回位标志[0001.04]
ANDNOT 801.07  ; #1腔体平移二级气缸伸出位标志[0001.07]
ORLD
ANDLD
OUT 406.02  ; #1-1电池注氦阀开[M]
LD TR0
LD 716.02  ; #1-1电池注氦阀关[SW]
OR D1077.01  ; #1腔体关闭除破真空阀以外全部阀门（复位）
ANDLD
DIFU(013) 316.02  ; #1-1电池注氦阀关[Pls]
LD TR0
LD 316.02  ; #1-1电池注氦阀关[Pls]
OR 416.02  ; #1-1电池注氦阀关[M]
ANDLD
ANDNOT 306.02  ; #1-1电池注氦阀开[Pls]
ANDNOT 823.01  ; #1-1电池注氦阀关到位标志
OUT 416.02  ; #1-1电池注氦阀关[M]

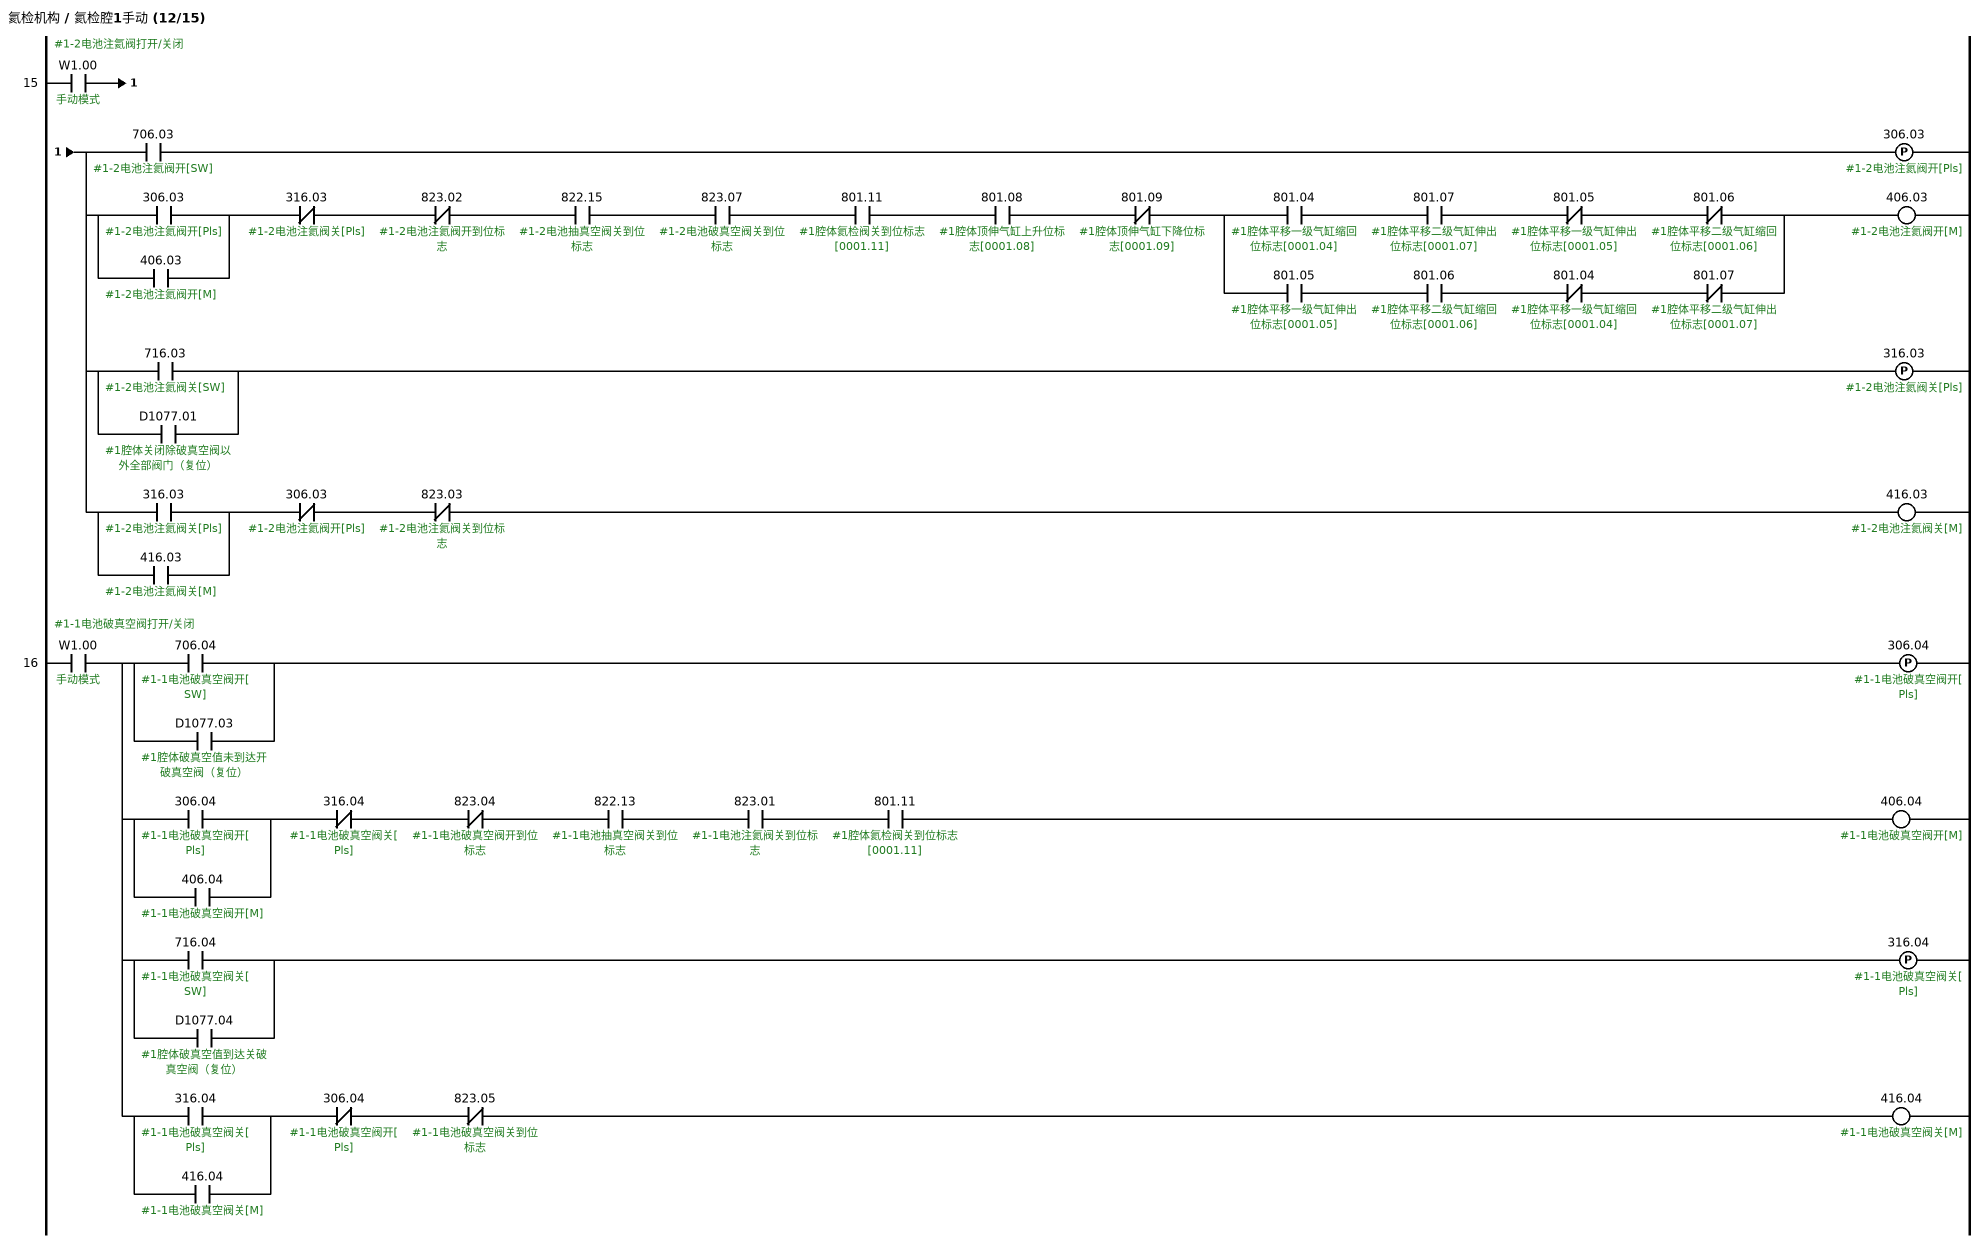
; rung 15: #1-2电池注氦阀打开/关闭
LD W1.00  ; 手动模式
OUT TR0
AND 706.03  ; #1-2电池注氦阀开[SW]
DIFU(013) 306.03  ; #1-2电池注氦阀开[Pls]
LD TR0
LD 306.03  ; #1-2电池注氦阀开[Pls]
OR 406.03  ; #1-2电池注氦阀开[M]
ANDLD
ANDNOT 316.03  ; #1-2电池注氦阀关[Pls]
ANDNOT 823.02  ; #1-2电池注氦阀开到位标志
AND 822.15  ; #1-2电池抽真空阀关到位标志
AND 823.07  ; #1-2电池破真空阀关到位标志
AND 801.11  ; #1腔体氦检阀关到位标志[0001.11]
AND 801.08  ; #1腔体顶伸气缸上升位标志[0001.08]
ANDNOT 801.09  ; #1腔体顶伸气缸下降位标志[0001.09]
LD 801.04  ; #1腔体平移一级气缸缩回位标志[0001.04]
AND 801.07  ; #1腔体平移二级气缸伸出位标志[0001.07]
ANDNOT 801.05  ; #1腔体平移一级气缸伸出位标志[0001.05]
ANDNOT 801.06  ; #1腔体平移二级气缸缩回位标志[0001.06]
LD 801.05  ; #1腔体平移一级气缸伸出位标志[0001.05]
AND 801.06  ; #1腔体平移二级气缸缩回位标志[0001.06]
ANDNOT 801.04  ; #1腔体平移一级气缸缩回位标志[0001.04]
ANDNOT 801.07  ; #1腔体平移二级气缸伸出位标志[0001.07]
ORLD
ANDLD
OUT 406.03  ; #1-2电池注氦阀开[M]
LD TR0
LD 716.03  ; #1-2电池注氦阀关[SW]
OR D1077.01  ; #1腔体关闭除破真空阀以外全部阀门（复位）
ANDLD
DIFU(013) 316.03  ; #1-2电池注氦阀关[Pls]
LD TR0
LD 316.03  ; #1-2电池注氦阀关[Pls]
OR 416.03  ; #1-2电池注氦阀关[M]
ANDLD
ANDNOT 306.03  ; #1-2电池注氦阀开[Pls]
ANDNOT 823.03  ; #1-2电池注氦阀关到位标志
OUT 416.03  ; #1-2电池注氦阀关[M]
; rung 16: #1-1电池破真空阀打开/关闭
LD W1.00  ; 手动模式
OUT TR0
LD 706.04  ; #1-1电池破真空阀开[SW]
OR D1077.03  ; #1腔体破真空值未到达开破真空阀（复位）
ANDLD
DIFU(013) 306.04  ; #1-1电池破真空阀开[Pls]
LD TR0
LD 306.04  ; #1-1电池破真空阀开[Pls]
OR 406.04  ; #1-1电池破真空阀开[M]
ANDLD
ANDNOT 316.04  ; #1-1电池破真空阀关[Pls]
ANDNOT 823.04  ; #1-1电池破真空阀开到位标志
AND 822.13  ; #1-1电池抽真空阀关到位标志
AND 823.01  ; #1-1电池注氦阀关到位标志
AND 801.11  ; #1腔体氦检阀关到位标志[0001.11]
OUT 406.04  ; #1-1电池破真空阀开[M]
LD TR0
LD 716.04  ; #1-1电池破真空阀关[SW]
OR D1077.04  ; #1腔体破真空值到达关破真空阀（复位）
ANDLD
DIFU(013) 316.04  ; #1-1电池破真空阀关[Pls]
LD TR0
LD 316.04  ; #1-1电池破真空阀关[Pls]
OR 416.04  ; #1-1电池破真空阀关[M]
ANDLD
ANDNOT 306.04  ; #1-1电池破真空阀开[Pls]
ANDNOT 823.05  ; #1-1电池破真空阀关到位标志
OUT 416.04  ; #1-1电池破真空阀关[M]

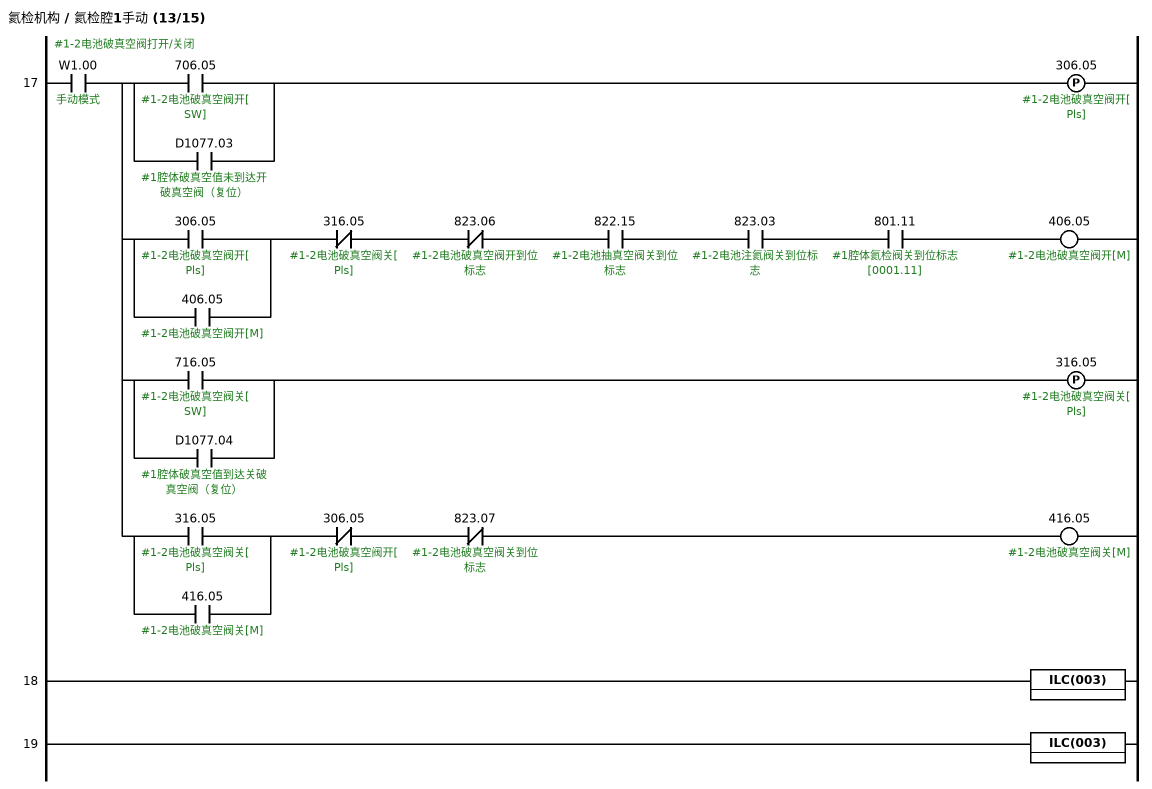
; rung 17: #1-2电池破真空阀打开/关闭
LD W1.00  ; 手动模式
OUT TR0
LD 706.05  ; #1-2电池破真空阀开[SW]
OR D1077.03  ; #1腔体破真空值未到达开破真空阀（复位）
ANDLD
DIFU(013) 306.05  ; #1-2电池破真空阀开[Pls]
LD TR0
LD 306.05  ; #1-2电池破真空阀开[Pls]
OR 406.05  ; #1-2电池破真空阀开[M]
ANDLD
ANDNOT 316.05  ; #1-2电池破真空阀关[Pls]
ANDNOT 823.06  ; #1-2电池破真空阀开到位标志
AND 822.15  ; #1-2电池抽真空阀关到位标志
AND 823.03  ; #1-2电池注氦阀关到位标志
AND 801.11  ; #1腔体氦检阀关到位标志[0001.11]
OUT 406.05  ; #1-2电池破真空阀开[M]
LD TR0
LD 716.05  ; #1-2电池破真空阀关[SW]
OR D1077.04  ; #1腔体破真空值到达关破真空阀（复位）
ANDLD
DIFU(013) 316.05  ; #1-2电池破真空阀关[Pls]
LD TR0
LD 316.05  ; #1-2电池破真空阀关[Pls]
OR 416.05  ; #1-2电池破真空阀关[M]
ANDLD
ANDNOT 306.05  ; #1-2电池破真空阀开[Pls]
ANDNOT 823.07  ; #1-2电池破真空阀关到位标志
OUT 416.05  ; #1-2电池破真空阀关[M]
; rung 18
ILC(003)
; rung 19
ILC(003)

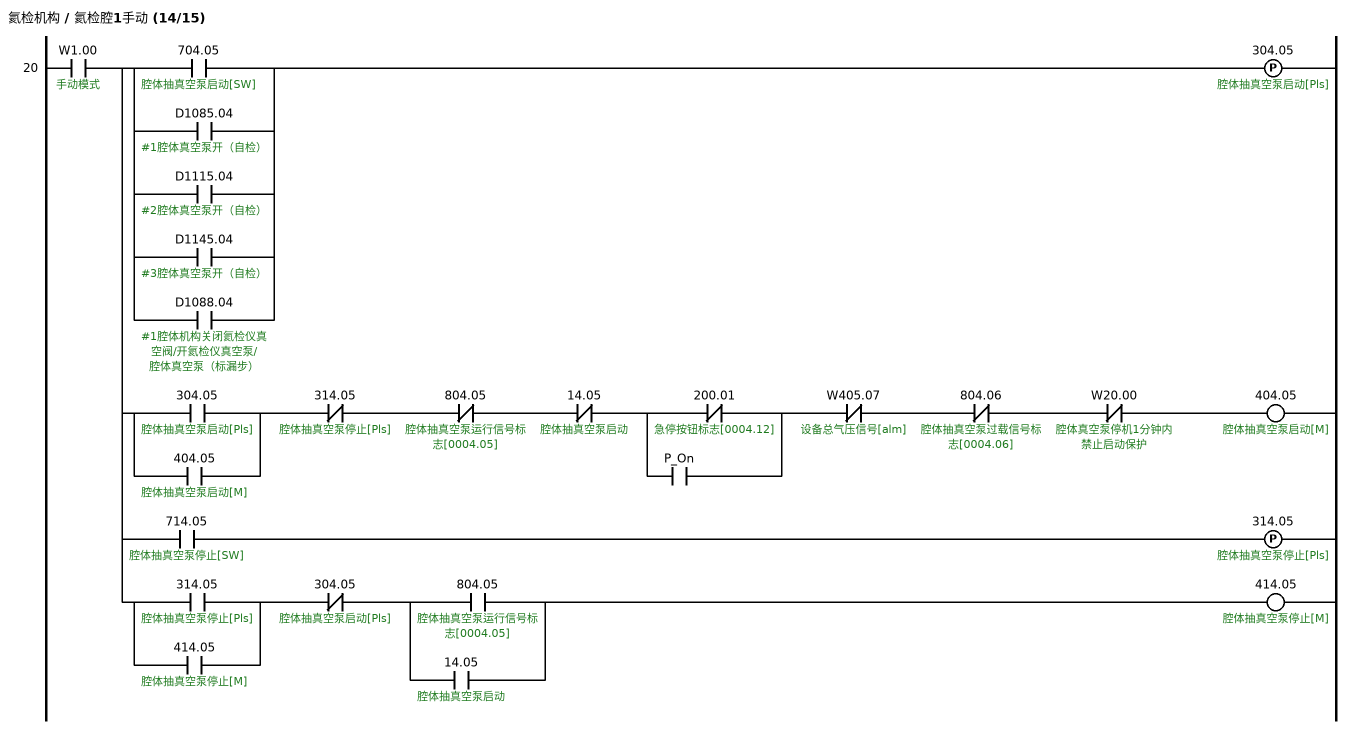
; rung 20
LD W1.00  ; 手动模式
OUT TR0
LD 704.05  ; 腔体抽真空泵启动[SW]
OR D1085.04  ; #1腔体真空泵开（自检）
OR D1115.04  ; #2腔体真空泵开（自检）
OR D1145.04  ; #3腔体真空泵开（自检）
OR D1088.04  ; #1腔体机构关闭氦检仪真空阀/开氦检仪真空泵/腔体真空泵（标漏步）
ANDLD
DIFU(013) 304.05  ; 腔体抽真空泵启动[Pls]
LD TR0
LD 304.05  ; 腔体抽真空泵启动[Pls]
OR 404.05  ; 腔体抽真空泵启动[M]
ANDLD
ANDNOT 314.05  ; 腔体抽真空泵停止[Pls]
ANDNOT 804.05  ; 腔体抽真空泵运行信号标志[0004.05]
ANDNOT 14.05  ; 腔体抽真空泵启动
LDNOT 200.01  ; 急停按钮标志[0004.12]
OR P_On
ANDLD
ANDNOT W405.07  ; 设备总气压信号[alm]
ANDNOT 804.06  ; 腔体抽真空泵过载信号标志[0004.06]
ANDNOT W20.00  ; 腔体真空泵停机1分钟内禁止启动保护
OUT 404.05  ; 腔体抽真空泵启动[M]
LD TR0
AND 714.05  ; 腔体抽真空泵停止[SW]
DIFU(013) 314.05  ; 腔体抽真空泵停止[Pls]
LD TR0
LD 314.05  ; 腔体抽真空泵停止[Pls]
OR 414.05  ; 腔体抽真空泵停止[M]
ANDLD
ANDNOT 304.05  ; 腔体抽真空泵启动[Pls]
LD 804.05  ; 腔体抽真空泵运行信号标志[0004.05]
OR 14.05  ; 腔体抽真空泵启动
ANDLD
OUT 414.05  ; 腔体抽真空泵停止[M]

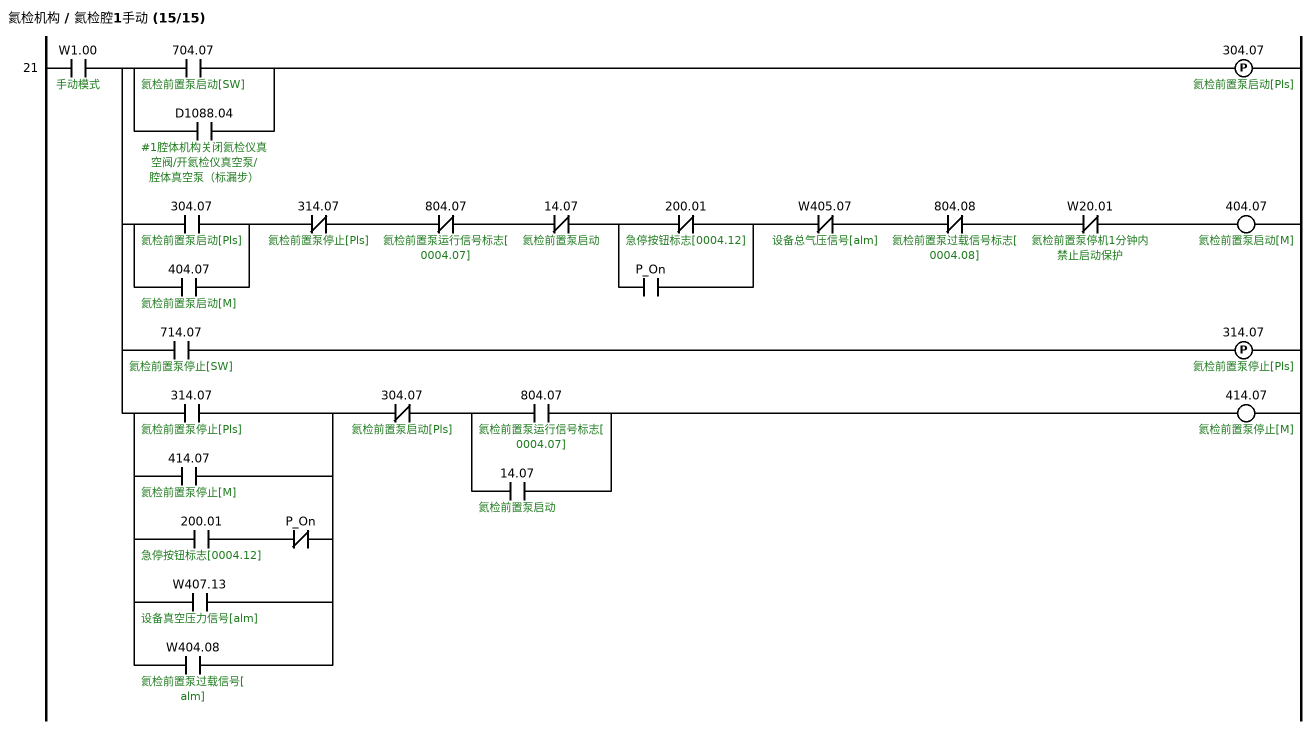
; rung 21
LD W1.00  ; 手动模式
OUT TR0
LD 704.07  ; 氦检前置泵启动[SW]
OR D1088.04  ; #1腔体机构关闭氦检仪真空阀/开氦检仪真空泵/腔体真空泵（标漏步）
ANDLD
DIFU(013) 304.07  ; 氦检前置泵启动[Pls]
LD TR0
LD 304.07  ; 氦检前置泵启动[Pls]
OR 404.07  ; 氦检前置泵启动[M]
ANDLD
ANDNOT 314.07  ; 氦检前置泵停止[Pls]
ANDNOT 804.07  ; 氦检前置泵运行信号标志[0004.07]
ANDNOT 14.07  ; 氦检前置泵启动
LDNOT 200.01  ; 急停按钮标志[0004.12]
OR P_On
ANDLD
ANDNOT W405.07  ; 设备总气压信号[alm]
ANDNOT 804.08  ; 氦检前置泵过载信号标志[0004.08]
ANDNOT W20.01  ; 氦检前置泵停机1分钟内禁止启动保护
OUT 404.07  ; 氦检前置泵启动[M]
LD TR0
AND 714.07  ; 氦检前置泵停止[SW]
DIFU(013) 314.07  ; 氦检前置泵停止[Pls]
LD TR0
LD 314.07  ; 氦检前置泵停止[Pls]
OR 414.07  ; 氦检前置泵停止[M]
LD 200.01  ; 急停按钮标志[0004.12]
ANDNOT P_On
ORLD
OR W407.13  ; 设备真空压力信号[alm]
OR W404.08  ; 氦检前置泵过载信号[alm]
ANDLD
ANDNOT 304.07  ; 氦检前置泵启动[Pls]
LD 804.07  ; 氦检前置泵运行信号标志[0004.07]
OR 14.07  ; 氦检前置泵启动
ANDLD
OUT 414.07  ; 氦检前置泵停止[M]

### Section 氦检腔2手动

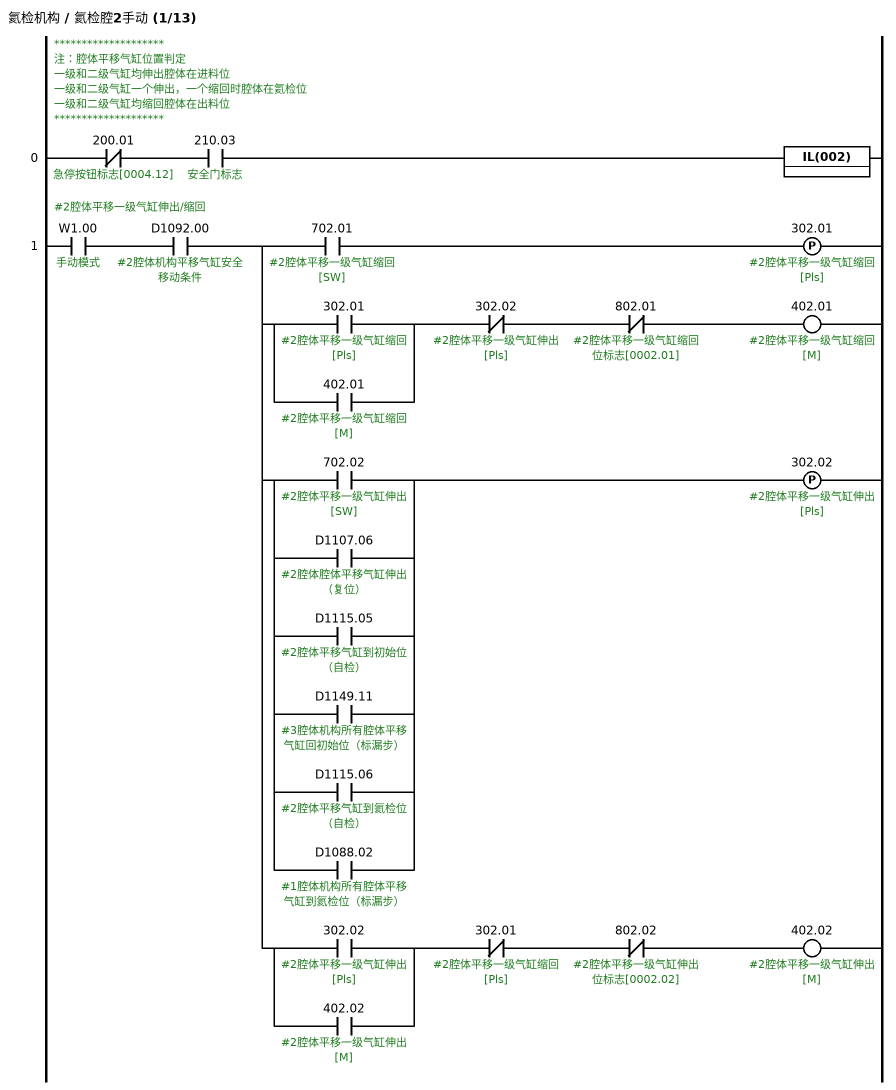
; rung 0: ******************** / 注：腔体平移气缸位置判定 / 一级和二级气缸均伸出腔体在进料位 / 一级和二级气缸一个伸出，一个缩回时腔体在氦检位 / 一级和二级气缸均缩回腔体在出料位 / ********************
LDNOT 200.01  ; 急停按钮标志[0004.12]
AND 210.03  ; 安全门标志
IL(002)
; rung 1: #2腔体平移一级气缸伸出/缩回
LD W1.00  ; 手动模式
AND D1092.00  ; #2腔体机构平移气缸安全移动条件
OUT TR0
AND 702.01  ; #2腔体平移一级气缸缩回[SW]
DIFU(013) 302.01  ; #2腔体平移一级气缸缩回[Pls]
LD TR0
LD 302.01  ; #2腔体平移一级气缸缩回[Pls]
OR 402.01  ; #2腔体平移一级气缸缩回[M]
ANDLD
ANDNOT 302.02  ; #2腔体平移一级气缸伸出[Pls]
ANDNOT 802.01  ; #2腔体平移一级气缸缩回位标志[0002.01]
OUT 402.01  ; #2腔体平移一级气缸缩回[M]
LD TR0
LD 702.02  ; #2腔体平移一级气缸伸出[SW]
OR D1107.06  ; #2腔体腔体平移气缸伸出（复位）
OR D1115.05  ; #2腔体平移气缸到初始位（自检）
OR D1149.11  ; #3腔体机构所有腔体平移气缸回初始位（标漏步）
OR D1115.06  ; #2腔体平移气缸到氦检位（自检）
OR D1088.02  ; #1腔体机构所有腔体平移气缸到氦检位（标漏步）
ANDLD
DIFU(013) 302.02  ; #2腔体平移一级气缸伸出[Pls]
LD TR0
LD 302.02  ; #2腔体平移一级气缸伸出[Pls]
OR 402.02  ; #2腔体平移一级气缸伸出[M]
ANDLD
ANDNOT 302.01  ; #2腔体平移一级气缸缩回[Pls]
ANDNOT 802.02  ; #2腔体平移一级气缸伸出位标志[0002.02]
OUT 402.02  ; #2腔体平移一级气缸伸出[M]

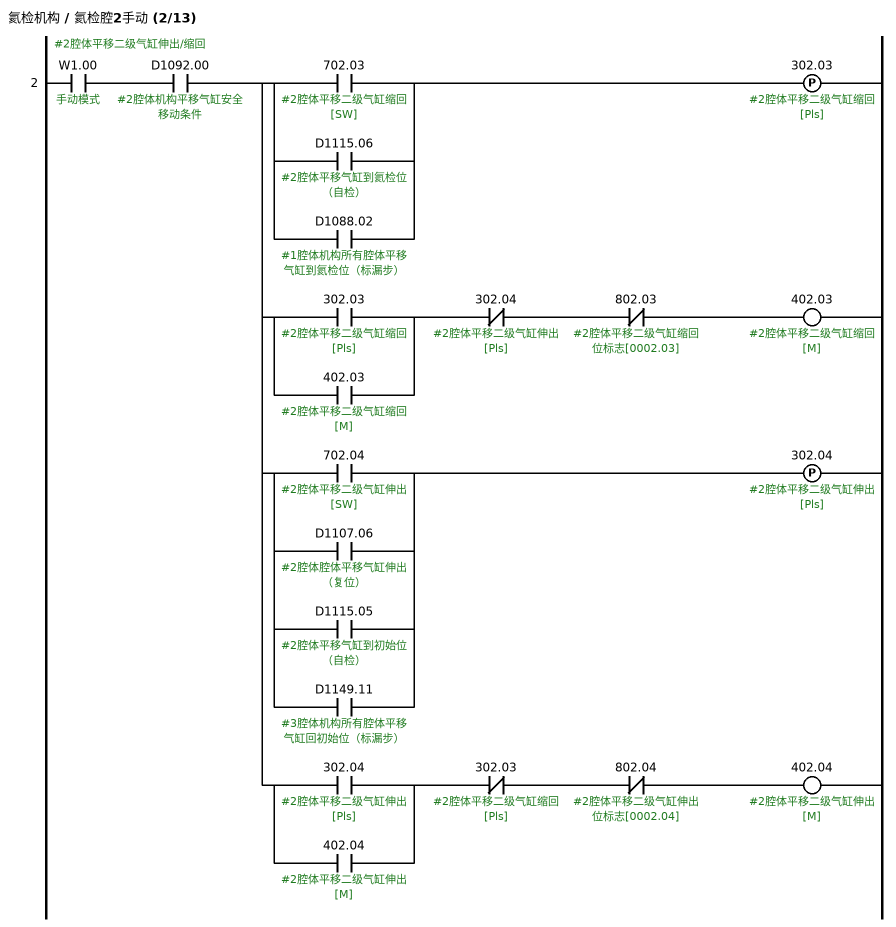
; rung 2: #2腔体平移二级气缸伸出/缩回
LD W1.00  ; 手动模式
AND D1092.00  ; #2腔体机构平移气缸安全移动条件
OUT TR0
LD 702.03  ; #2腔体平移二级气缸缩回[SW]
OR D1115.06  ; #2腔体平移气缸到氦检位（自检）
OR D1088.02  ; #1腔体机构所有腔体平移气缸到氦检位（标漏步）
ANDLD
DIFU(013) 302.03  ; #2腔体平移二级气缸缩回[Pls]
LD TR0
LD 302.03  ; #2腔体平移二级气缸缩回[Pls]
OR 402.03  ; #2腔体平移二级气缸缩回[M]
ANDLD
ANDNOT 302.04  ; #2腔体平移二级气缸伸出[Pls]
ANDNOT 802.03  ; #2腔体平移二级气缸缩回位标志[0002.03]
OUT 402.03  ; #2腔体平移二级气缸缩回[M]
LD TR0
LD 702.04  ; #2腔体平移二级气缸伸出[SW]
OR D1107.06  ; #2腔体腔体平移气缸伸出（复位）
OR D1115.05  ; #2腔体平移气缸到初始位（自检）
OR D1149.11  ; #3腔体机构所有腔体平移气缸回初始位（标漏步）
ANDLD
DIFU(013) 302.04  ; #2腔体平移二级气缸伸出[Pls]
LD TR0
LD 302.04  ; #2腔体平移二级气缸伸出[Pls]
OR 402.04  ; #2腔体平移二级气缸伸出[M]
ANDLD
ANDNOT 302.03  ; #2腔体平移二级气缸缩回[Pls]
ANDNOT 802.04  ; #2腔体平移二级气缸伸出位标志[0002.04]
OUT 402.04  ; #2腔体平移二级气缸伸出[M]

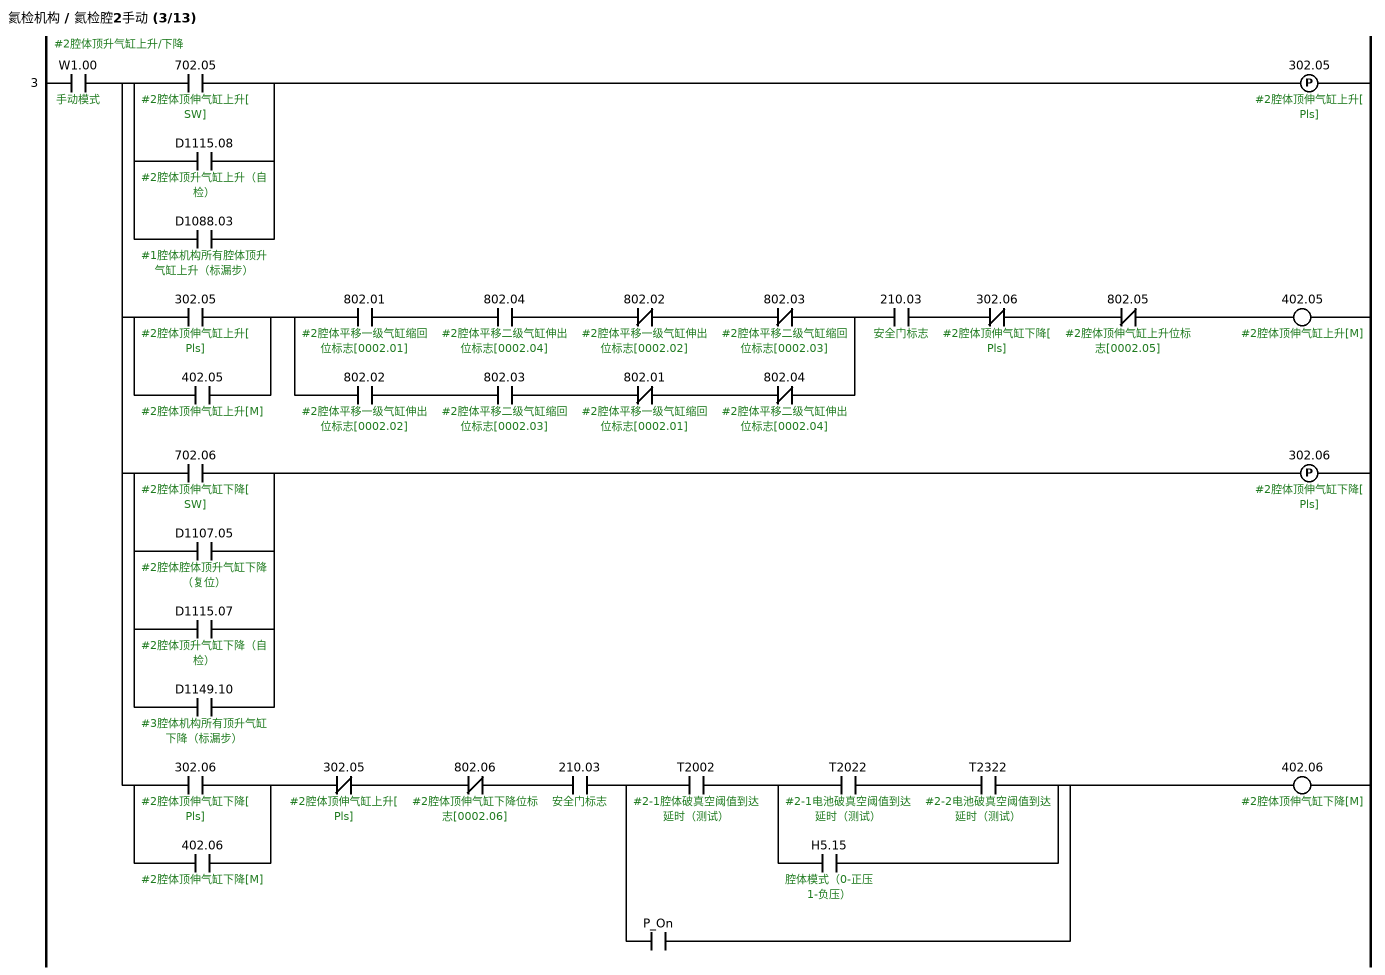
; rung 3: #2腔体顶升气缸上升/下降
LD W1.00  ; 手动模式
OUT TR0
LD 702.05  ; #2腔体顶伸气缸上升[SW]
OR D1115.08  ; #2腔体顶升气缸上升（自检）
OR D1088.03  ; #1腔体机构所有腔体顶升气缸上升（标漏步）
ANDLD
DIFU(013) 302.05  ; #2腔体顶伸气缸上升[Pls]
LD TR0
LD 302.05  ; #2腔体顶伸气缸上升[Pls]
OR 402.05  ; #2腔体顶伸气缸上升[M]
ANDLD
LD 802.01  ; #2腔体平移一级气缸缩回位标志[0002.01]
AND 802.04  ; #2腔体平移二级气缸伸出位标志[0002.04]
ANDNOT 802.02  ; #2腔体平移一级气缸伸出位标志[0002.02]
ANDNOT 802.03  ; #2腔体平移二级气缸缩回位标志[0002.03]
LD 802.02  ; #2腔体平移一级气缸伸出位标志[0002.02]
AND 802.03  ; #2腔体平移二级气缸缩回位标志[0002.03]
ANDNOT 802.01  ; #2腔体平移一级气缸缩回位标志[0002.01]
ANDNOT 802.04  ; #2腔体平移二级气缸伸出位标志[0002.04]
ORLD
ANDLD
AND 210.03  ; 安全门标志
ANDNOT 302.06  ; #2腔体顶伸气缸下降[Pls]
ANDNOT 802.05  ; #2腔体顶伸气缸上升位标志[0002.05]
OUT 402.05  ; #2腔体顶伸气缸上升[M]
LD TR0
LD 702.06  ; #2腔体顶伸气缸下降[SW]
OR D1107.05  ; #2腔体腔体顶升气缸下降（复位）
OR D1115.07  ; #2腔体顶升气缸下降（自检）
OR D1149.10  ; #3腔体机构所有顶升气缸下降（标漏步）
ANDLD
DIFU(013) 302.06  ; #2腔体顶伸气缸下降[Pls]
LD TR0
LD 302.06  ; #2腔体顶伸气缸下降[Pls]
OR 402.06  ; #2腔体顶伸气缸下降[M]
ANDLD
ANDNOT 302.05  ; #2腔体顶伸气缸上升[Pls]
ANDNOT 802.06  ; #2腔体顶伸气缸下降位标志[0002.06]
AND 210.03  ; 安全门标志
LD T2002  ; #2-1腔体破真空阈值到达延时（测试）
LD T2022  ; #2-1电池破真空阈值到达延时（测试）
AND T2322  ; #2-2电池破真空阈值到达延时（测试）
OR H5.15  ; 腔体模式（0-正压 1-负压）
ANDLD
OR P_On
ANDLD
OUT 402.06  ; #2腔体顶伸气缸下降[M]

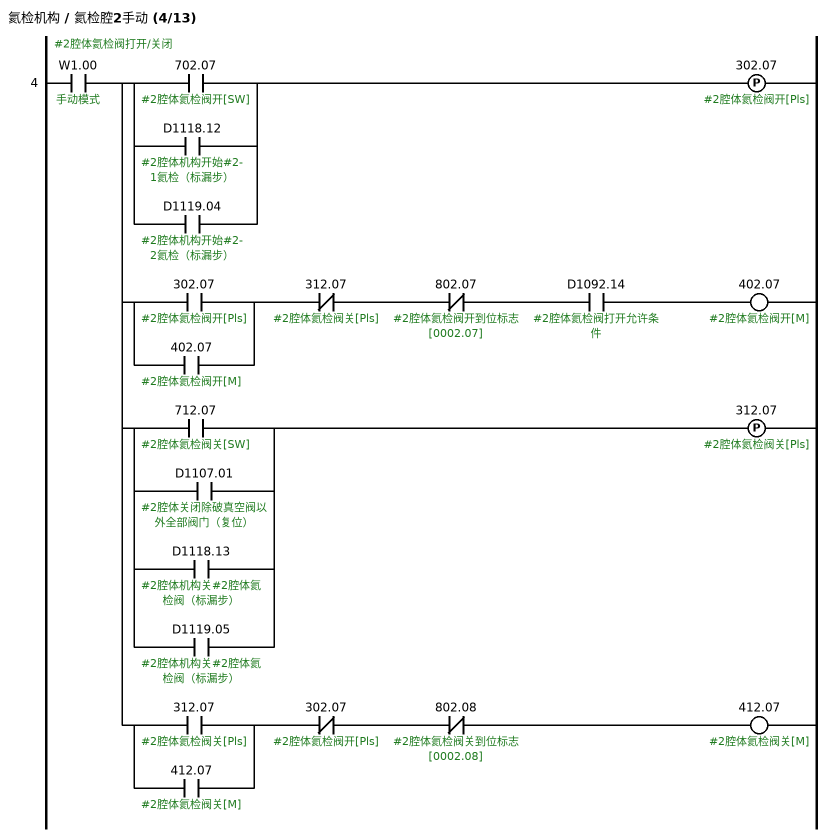
; rung 4: #2腔体氦检阀打开/关闭
LD W1.00  ; 手动模式
OUT TR0
LD 702.07  ; #2腔体氦检阀开[SW]
OR D1118.12  ; #2腔体机构开始#2-1氦检（标漏步）
OR D1119.04  ; #2腔体机构开始#2-2氦检（标漏步）
ANDLD
DIFU(013) 302.07  ; #2腔体氦检阀开[Pls]
LD TR0
LD 302.07  ; #2腔体氦检阀开[Pls]
OR 402.07  ; #2腔体氦检阀开[M]
ANDLD
ANDNOT 312.07  ; #2腔体氦检阀关[Pls]
ANDNOT 802.07  ; #2腔体氦检阀开到位标志[0002.07]
AND D1092.14  ; #2腔体氦检阀打开允许条件
OUT 402.07  ; #2腔体氦检阀开[M]
LD TR0
LD 712.07  ; #2腔体氦检阀关[SW]
OR D1107.01  ; #2腔体关闭除破真空阀以外全部阀门（复位）
OR D1118.13  ; #2腔体机构关#2腔体氦检阀（标漏步）
OR D1119.05  ; #2腔体机构关#2腔体氦检阀（标漏步）
ANDLD
DIFU(013) 312.07  ; #2腔体氦检阀关[Pls]
LD TR0
LD 312.07  ; #2腔体氦检阀关[Pls]
OR 412.07  ; #2腔体氦检阀关[M]
ANDLD
ANDNOT 302.07  ; #2腔体氦检阀开[Pls]
ANDNOT 802.08  ; #2腔体氦检阀关到位标志[0002.08]
OUT 412.07  ; #2腔体氦检阀关[M]

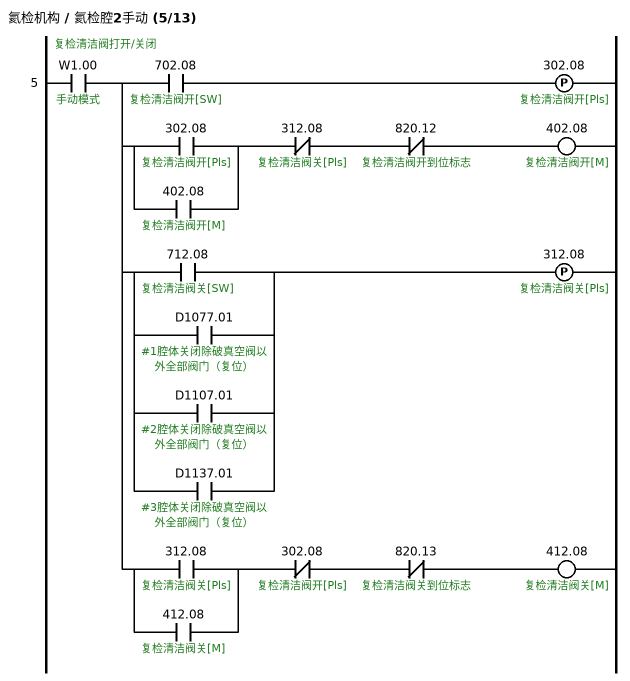
; rung 5: 复检清洁阀打开/关闭
LD W1.00  ; 手动模式
OUT TR0
AND 702.08  ; 复检清洁阀开[SW]
DIFU(013) 302.08  ; 复检清洁阀开[Pls]
LD TR0
LD 302.08  ; 复检清洁阀开[Pls]
OR 402.08  ; 复检清洁阀开[M]
ANDLD
ANDNOT 312.08  ; 复检清洁阀关[Pls]
ANDNOT 820.12  ; 复检清洁阀开到位标志
OUT 402.08  ; 复检清洁阀开[M]
LD TR0
LD 712.08  ; 复检清洁阀关[SW]
OR D1077.01  ; #1腔体关闭除破真空阀以外全部阀门（复位）
OR D1107.01  ; #2腔体关闭除破真空阀以外全部阀门（复位）
OR D1137.01  ; #3腔体关闭除破真空阀以外全部阀门（复位）
ANDLD
DIFU(013) 312.08  ; 复检清洁阀关[Pls]
LD TR0
LD 312.08  ; 复检清洁阀关[Pls]
OR 412.08  ; 复检清洁阀关[M]
ANDLD
ANDNOT 302.08  ; 复检清洁阀开[Pls]
ANDNOT 820.13  ; 复检清洁阀关到位标志
OUT 412.08  ; 复检清洁阀关[M]

